LIN {X 0,Y 573.119,Z 536.24,A -85,B 0,C 180,E1 -2257.22,E2 -2257.22} C_VEL
LIN {X 0,Y 573.2,Z 527.994,A -85,B 0,C 180,E1 -2258.283,E2 -2258.283} C_VEL
LIN {X 0,Y 573.286,Z 519.543,A -85,B 0,C 180,E1 -2259.17,E2 -2259.17} C_VEL
LIN {X 0,Y 573.411,Z 509.104,A -85,B 0,C 180,E1 -2260.058,E2 -2260.058} C_VEL
LIN {X 0,Y 573.557,Z 497.409,A -85,B 0,C 180,E1 -2260.854,E2 -2260.854} C_VEL
LIN {X 0,Y 573.652,Z 486.296,A -85,B 0,C 180,E1 -2261.447,E2 -2261.447} C_VEL
LIN {X 0,Y 573.693,Z 474.485,A -85,B 0,C 180,E1 -2261.93,E2 -2261.93} C_VEL
LIN {X 0,Y 573.817,Z 461.452,A -85,B 0,C 180,E1 -2262.309,E2 -2262.309} C_VEL
LIN {X 0,Y 573.865,Z 449.117,A -85,B 0,C 180,E1 -2262.532,E2 -2262.532} C_VEL
LIN {X 0,Y 573.918,Z 350.087,A -85,B 0,C 180,E1 -2263.778,E2 -2263.778} C_VEL
LIN {X 0,Y 573.419,Z 346.442,A -85,B 0,C 180,E1 -2263.85,E2 -2263.85} C_VEL
LIN {X 0,Y 573.59,Z 325.392,A -85,B 0,C 180,E1 -2266.726,E2 -2266.726} C_VEL
LIN {X 0,Y 573.813,Z 304.327,A -85,B 0,C 180,E1 -2269.645,E2 -2269.645} C_VEL
LIN {X 0,Y 574.01,Z 285.256,A -85,B 0,C 180,E1 -2272.306,E2 -2272.306} C_VEL
LIN {X 0,Y 574.012,Z 277.944,A -85,B 0,C 180,E1 -2273.325,E2 -2273.325} C_VEL
LIN {X 0,Y 573.226,Z 274.085,A -85,B 0,C 180,E1 -2273.913,E2 -2273.913} C_VEL
LIN {X 0,Y 573.199,Z 274.087,A -85,B 0,C 180,E1 -2276.484,E2 -2276.484} C_VEL
LIN {X 0,Y 573.238,Z 274.076,A -85,B 0,C 180,E1 -2279.367,E2 -2279.367} C_VEL
LIN {X 0,Y 573.248,Z 274.082,A -85,B 0,C 180,E1 -2282.227,E2 -2282.227} C_VEL
LIN {X 0,Y 573.202,Z 274.08,A -85,B 0,C 180,E1 -2285.188,E2 -2285.188} C_VEL
LIN {X 0,Y 573.227,Z 274.077,A -85,B 0,C 180,E1 -2287.808,E2 -2287.808} C_VEL
LIN {X 0,Y 573.243,Z 274.082,A -85,B 0,C 180,E1 -2290.525,E2 -2290.525} C_VEL
LIN {X 0,Y 573.229,Z 274.075,A -85,B 0,C 180,E1 -2293.359,E2 -2293.359} C_VEL
LIN {X 0,Y 573.236,Z 274.082,A -85,B 0,C 180,E1 -2296.331,E2 -2296.331} C_VEL
LIN {X 0,Y 573.226,Z 274.085,A -85,B 0,C 180,E1 -2298.543,E2 -2298.543} C_VEL
LIN {X 0,Y 573.241,Z 274.074,A -85,B 0,C 180,E1 -2301.298,E2 -2301.298} C_VEL
LIN {X 0,Y 573.211,Z 274.079,A -85,B 0,C 180,E1 -2304.018,E2 -2304.018} C_VEL
LIN {X 0,Y 573.236,Z 274.083,A -85,B 0,C 180,E1 -2306.516,E2 -2306.516} C_VEL
LIN {X 0,Y 573.229,Z 274.077,A -85,B 0,C 180,E1 -2309.117,E2 -2309.117} C_VEL
LIN {X 0,Y 573.248,Z 274.073,A -85,B 0,C 180,E1 -2311.971,E2 -2311.971} C_VEL
LIN {X 0,Y 573.245,Z 274.082,A -85,B 0,C 180,E1 -2314.59,E2 -2314.59} C_VEL
LIN {X 0,Y 573.234,Z 274.074,A -85,B 0,C 180,E1 -2317.662,E2 -2317.662} C_VEL
LIN {X 0,Y 573.276,Z 274.079,A -85,B 0,C 180,E1 -2320.728,E2 -2320.728} C_VEL
LIN {X 0,Y 573.256,Z 274.071,A -85,B 0,C 180,E1 -2323.622,E2 -2323.622} C_VEL
LIN {X 0,Y 573.235,Z 274.08,A -85,B 0,C 180,E1 -2326.53,E2 -2326.53} C_VEL
LIN {X 0,Y 573.26,Z 274.08,A -85,B 0,C 180,E1 -2328.745,E2 -2328.745} C_VEL
LIN {X 0,Y 573.282,Z 274.068,A -85,B 0,C 180,E1 -2331.541,E2 -2331.541} C_VEL
LIN {X 0,Y 573.288,Z 274.07,A -85,B 0,C 180,E1 -2334.372,E2 -2334.372} C_VEL
LIN {X 0,Y 573.31,Z 274.065,A -85,B 0,C 180,E1 -2337.893,E2 -2337.893} C_VEL
LIN {X 0,Y 573.33,Z 274.068,A -85,B 0,C 180,E1 -2340.703,E2 -2340.703} C_VEL
LIN {X 0,Y 573.303,Z 274.074,A -85,B 0,C 180,E1 -2342.811,E2 -2342.811} C_VEL
LIN {X 0,Y 573.286,Z 274.069,A -85,B 0,C 180,E1 -2345.628,E2 -2345.628} C_VEL
LIN {X 0,Y 573.286,Z 274.07,A -85,B 0,C 180,E1 -2348.46,E2 -2348.46} C_VEL
LIN {X 0,Y 573.269,Z 274.076,A -85,B 0,C 180,E1 -2351.312,E2 -2351.312} C_VEL
LIN {X 0,Y 573.279,Z 274.069,A -85,B 0,C 180,E1 -2354.425,E2 -2354.425} C_VEL
LIN {X 0,Y 573.256,Z 274.081,A -85,B 0,C 180,E1 -2357.112,E2 -2357.112} C_VEL
LIN {X 0,Y 573.24,Z 274.073,A -85,B 0,C 180,E1 -2360.077,E2 -2360.077} C_VEL
LIN {X 0,Y 573.231,Z 274.075,A -85,B 0,C 180,E1 -2362.338,E2 -2362.338} C_VEL
LIN {X 0,Y 573.243,Z 274.074,A -85,B 0,C 180,E1 -2364.388,E2 -2364.388} C_VEL
LIN {X 0,Y 572.622,Z 274.158,A -85,B 0,C 180,E1 -2364.974,E2 -2364.974} C_VEL
LIN {X 0,Y 569.784,Z 274.516,A -85,B 0,C 180,E1 -2365.926,E2 -2365.926} C_VEL
LIN {X 0,Y 567.35,Z 274.82,A -85,B 0,C 180,E1 -2366.691,E2 -2366.691} C_VEL
LIN {X 0,Y 566.288,Z 274.949,A -85,B 0,C 180,E1 -2367.282,E2 -2367.282} C_VEL
LIN {X 0,Y 566.195,Z 274.957,A -85,B 0,C 180,E1 -2367.483,E2 -2367.483} C_VEL
LIN {X 0,Y 566.194,Z 274.954,A -85,B 0,C 180,E1 -2369.77,E2 -2369.77} C_VEL
LIN {X 0,Y 566.199,Z 274.95,A -85,B 0,C 180,E1 -2372.43,E2 -2372.43} C_VEL
LIN {X 0,Y 566.193,Z 274.957,A -85,B 0,C 180,E1 -2374.992,E2 -2374.992} C_VEL
LIN {X 0,Y 566.194,Z 274.958,A -85,B 0,C 180,E1 -2377.462,E2 -2377.462} C_VEL
LIN {X 0,Y 566.205,Z 274.95,A -85,B 0,C 180,E1 -2380.2,E2 -2380.2} C_VEL
LIN {X 0,Y 566.18,Z 274.958,A -85,B 0,C 180,E1 -2383.057,E2 -2383.057} C_VEL
LIN {X 0,Y 566.157,Z 274.958,A -85,B 0,C 180,E1 -2386.054,E2 -2386.054} C_VEL
LIN {X 0,Y 566.157,Z 274.958,A -85,B 0,C 180,E1 -2388.859,E2 -2388.859} C_VEL
LIN {X 0,Y 566.201,Z 274.961,A -85,B 0,C 180,E1 -2391.444,E2 -2391.444} C_VEL
LIN {X 0,Y 566.143,Z 274.958,A -85,B 0,C 180,E1 -2394.307,E2 -2394.307} C_VEL
LIN {X 0,Y 566.194,Z 274.954,A -85,B 0,C 180,E1 -2396.897,E2 -2396.897} C_VEL
LIN {X 0,Y 566.166,Z 274.964,A -85,B 0,C 180,E1 -2399.407,E2 -2399.407} C_VEL
LIN {X 0,Y 566.198,Z 274.956,A -85,B 0,C 180,E1 -2402.586,E2 -2402.586} C_VEL
LIN {X 0,Y 566.328,Z 280.666,A -85,B 0,C 180,E1 -2403.664,E2 -2403.664} C_VEL
LIN {X 0,Y 566.236,Z 295.178,A -85,B 0,C 180,E1 -2406.405,E2 -2406.405} C_VEL
LIN {X 0,Y 566.225,Z 298.604,A -85,B 0,C 180,E1 -2407.047,E2 -2407.047} C_VEL
LIN {X 0,Y 567.18,Z 304.563,A -85,B 0,C 180,E1 -2407.157,E2 -2407.157} C_VEL
LIN {X 0,Y 566.919,Z 405.543,A -85,B 0,C 180,E1 -2408.459,E2 -2408.459} C_VEL
LIN {X 0,Y 566.843,Z 419.197,A -85,B 0,C 180,E1 -2408.793,E2 -2408.793} C_VEL
LIN {X 0,Y 566.723,Z 431.898,A -85,B 0,C 180,E1 -2409.256,E2 -2409.256} C_VEL
LIN {X 0,Y 566.555,Z 444.148,A -85,B 0,C 180,E1 -2409.865,E2 -2409.865} C_VEL
LIN {X 0,Y 566.418,Z 455.088,A -85,B 0,C 180,E1 -2410.562,E2 -2410.562} C_VEL
LIN {X 0,Y 566.299,Z 465.233,A -85,B 0,C 180,E1 -2411.364,E2 -2411.364} C_VEL
LIN {X 0,Y 566.183,Z 474.756,A -85,B 0,C 180,E1 -2412.295,E2 -2412.295} C_VEL
LIN {X 0,Y 566.05,Z 483.938,A -85,B 0,C 180,E1 -2413.408,E2 -2413.408} C_VEL
LIN {X 0,Y 566.009,Z 491.238,A -85,B 0,C 180,E1 -2414.517,E2 -2414.517} C_VEL
LIN {X 0,Y 565.941,Z 496.998,A -85,B 0,C 180,E1 -2415.62,E2 -2415.62} C_VEL
LIN {X 0,Y 565.928,Z 501.492,A -85,B 0,C 180,E1 -2416.719,E2 -2416.719} C_VEL
LIN {X 0,Y 565.894,Z 504.853,A -85,B 0,C 180,E1 -2417.812,E2 -2417.812} C_VEL
LIN {X 0,Y 565.904,Z 507.1,A -85,B 0,C 180,E1 -2418.847,E2 -2418.847} C_VEL
LIN {X 0,Y 565.882,Z 508.554,A -85,B 0,C 180,E1 -2419.987,E2 -2419.987} C_VEL
LIN {X 0,Y 565.852,Z 508.921,A -85,B 0,C 180,E1 -2421.429,E2 -2421.429} C_VEL
LIN {X 0,Y 565.879,Z 508.522,A -85,B 0,C 180,E1 -2422.148,E2 -2422.148} C_VEL
LIN {X 0,Y 565.921,Z 506.681,A -85,B 0,C 180,E1 -2423.466,E2 -2423.466} C_VEL
LIN {X 0,Y 565.916,Z 503.806,A -85,B 0,C 180,E1 -2424.656,E2 -2424.656} C_VEL
LIN {X 0,Y 565.957,Z 500.162,A -85,B 0,C 180,E1 -2425.728,E2 -2425.728} C_VEL
LIN {X 0,Y 565.954,Z 495.423,A -85,B 0,C 180,E1 -2426.797,E2 -2426.797} C_VEL
LIN {X 0,Y 566.008,Z 488.339,A -85,B 0,C 180,E1 -2428.044,E2 -2428.044} C_VEL
LIN {X 0,Y 566.12,Z 480.648,A -85,B 0,C 180,E1 -2429.111,E2 -2429.111} C_VEL
LIN {X 0,Y 566.205,Z 471.063,A -85,B 0,C 180,E1 -2430.178,E2 -2430.178} C_VEL
LIN {X 0,Y 566.328,Z 461.195,A -85,B 0,C 180,E1 -2431.067,E2 -2431.067} C_VEL
LIN {X 0,Y 566.445,Z 450.086,A -85,B 0,C 180,E1 -2431.867,E2 -2431.867} C_VEL
LIN {X 0,Y 566.588,Z 439.243,A -85,B 0,C 180,E1 -2432.489,E2 -2432.489} C_VEL
LIN {X 0,Y 566.702,Z 427.292,A -85,B 0,C 180,E1 -2433.022,E2 -2433.022} C_VEL
LIN {X 0,Y 566.816,Z 414.954,A -85,B 0,C 180,E1 -2433.421,E2 -2433.421} C_VEL
LIN {X 0,Y 566.89,Z 402.186,A -85,B 0,C 180,E1 -2433.688,E2 -2433.688} C_VEL
LIN {X 0,Y 567.102,Z 303.98,A -85,B 0,C 180,E1 -2434.942,E2 -2434.942} C_VEL
LIN {X 0,Y 566.257,Z 298.554,A -85,B 0,C 180,E1 -2435.051,E2 -2435.051} C_VEL
LIN {X 0,Y 566.353,Z 283.716,A -85,B 0,C 180,E1 -2437.846,E2 -2437.846} C_VEL
LIN {X 0,Y 566.213,Z 275.181,A -85,B 0,C 180,E1 -2439.466,E2 -2439.466} C_VEL
LIN {X 0,Y 566.169,Z 274.959,A -85,B 0,C 180,E1 -2439.648,E2 -2439.648} C_VEL
LIN {X 0,Y 566.185,Z 274.958,A -85,B 0,C 180,E1 -2442.183,E2 -2442.183} C_VEL
LIN {X 0,Y 566.194,Z 274.954,A -85,B 0,C 180,E1 -2445.11,E2 -2445.11} C_VEL
LIN {X 0,Y 566.175,Z 274.955,A -85,B 0,C 180,E1 -2448.079,E2 -2448.079} C_VEL
LIN {X 0,Y 566.208,Z 274.953,A -85,B 0,C 180,E1 -2450.338,E2 -2450.338} C_VEL
LIN {X 0,Y 566.171,Z 274.957,A -85,B 0,C 180,E1 -2453.28,E2 -2453.28} C_VEL
LIN {X 0,Y 566.178,Z 274.953,A -85,B 0,C 180,E1 -2455.751,E2 -2455.751} C_VEL
LIN {X 0,Y 566.157,Z 274.956,A -85,B 0,C 180,E1 -2458.192,E2 -2458.192} C_VEL
LIN {X 0,Y 566.182,Z 274.962,A -85,B 0,C 180,E1 -2461.074,E2 -2461.074} C_VEL
LIN {X 0,Y 566.202,Z 274.951,A -85,B 0,C 180,E1 -2463.732,E2 -2463.732} C_VEL
LIN {X 0,Y 566.185,Z 274.954,A -85,B 0,C 180,E1 -2466.572,E2 -2466.572} C_VEL
LIN {X 0,Y 566.21,Z 274.952,A -85,B 0,C 180,E1 -2469.684,E2 -2469.684} C_VEL
LIN {X 0,Y 566.183,Z 274.959,A -85,B 0,C 180,E1 -2473.056,E2 -2473.056} C_VEL
LIN {X 0,Y 566.16,Z 274.956,A -85,B 0,C 180,E1 -2476.053,E2 -2476.053} C_VEL
LIN {X 0,Y 566.159,Z 274.958,A -85,B 0,C 180,E1 -2478.858,E2 -2478.858} C_VEL
LIN {X 0,Y 566.203,Z 274.961,A -85,B 0,C 180,E1 -2481.444,E2 -2481.444} C_VEL
LIN {X 0,Y 566.146,Z 274.957,A -85,B 0,C 180,E1 -2484.306,E2 -2484.306} C_VEL
LIN {X 0,Y 566.199,Z 274.951,A -85,B 0,C 180,E1 -2486.896,E2 -2486.896} C_VEL
LIN {X 0,Y 566.171,Z 274.961,A -85,B 0,C 180,E1 -2489.406,E2 -2489.406} C_VEL
LIN {X 0,Y 566.193,Z 274.959,A -85,B 0,C 180,E1 -2491.856,E2 -2491.856} C_VEL
LIN {X 0,Y 566.183,Z 274.953,A -85,B 0,C 180,E1 -2494.979,E2 -2494.979} C_VEL
LIN {X 0,Y 566.191,Z 274.956,A -85,B 0,C 180,E1 -2498.137,E2 -2498.137} C_VEL
LIN {X 0,Y 566.236,Z 274.946,A -85,B 0,C 180,E1 -2500.614,E2 -2500.614} C_VEL
LIN {X 0,Y 566.169,Z 274.957,A -85,B 0,C 180,E1 -2503.411,E2 -2503.411} C_VEL
LIN {X 0,Y 566.226,Z 274.952,A -85,B 0,C 180,E1 -2505.626,E2 -2505.626} C_VEL
LIN {X 0,Y 566.194,Z 274.952,A -85,B 0,C 180,E1 -2508.699,E2 -2508.699} C_VEL
LIN {X 0,Y 566.198,Z 274.952,A -85,B 0,C 180,E1 -2511.434,E2 -2511.434} C_VEL
LIN {X 0,Y 566.242,Z 274.953,A -85,B 0,C 180,E1 -2514.301,E2 -2514.301} C_VEL
LIN {X 0,Y 566.279,Z 274.945,A -85,B 0,C 180,E1 -2517.866,E2 -2517.866} C_VEL
LIN {X 0,Y 566.289,Z 274.943,A -85,B 0,C 180,E1 -2520.711,E2 -2520.711} C_VEL
LIN {X 0,Y 566.249,Z 274.947,A -85,B 0,C 180,E1 -2522.846,E2 -2522.846} C_VEL
LIN {X 0,Y 566.232,Z 274.947,A -85,B 0,C 180,E1 -2525.698,E2 -2525.698} C_VEL
LIN {X 0,Y 566.192,Z 274.96,A -85,B 0,C 180,E1 -2528.566,E2 -2528.566} C_VEL
LIN {X 0,Y 566.197,Z 274.951,A -85,B 0,C 180,E1 -2531.455,E2 -2531.455} C_VEL
LIN {X 0,Y 566.218,Z 274.957,A -85,B 0,C 180,E1 -2534.498,E2 -2534.498} C_VEL
LIN {X 0,Y 566.176,Z 274.954,A -85,B 0,C 180,E1 -2537.332,E2 -2537.332} C_VEL
LIN {X 0,Y 566.205,Z 274.954,A -85,B 0,C 180,E1 -2540.337,E2 -2540.337} C_VEL
LIN {X 0,Y 566.169,Z 274.957,A -85,B 0,C 180,E1 -2543.279,E2 -2543.279} C_VEL
LIN {X 0,Y 566.174,Z 274.953,A -85,B 0,C 180,E1 -2545.751,E2 -2545.751} C_VEL
LIN {X 0,Y 566.154,Z 274.957,A -85,B 0,C 180,E1 -2548.192,E2 -2548.192} C_VEL
LIN {X 0,Y 566.179,Z 274.962,A -85,B 0,C 180,E1 -2551.073,E2 -2551.073} C_VEL
LIN {X 0,Y 566.199,Z 274.951,A -85,B 0,C 180,E1 -2553.731,E2 -2553.731} C_VEL
LIN {X 0,Y 566.183,Z 274.955,A -85,B 0,C 180,E1 -2556.571,E2 -2556.571} C_VEL
LIN {X 0,Y 566.208,Z 274.952,A -85,B 0,C 180,E1 -2559.684,E2 -2559.684} C_VEL
LIN {X 0,Y 566.181,Z 274.96,A -85,B 0,C 180,E1 -2563.056,E2 -2563.056} C_VEL
LIN {X 0,Y 566.158,Z 274.956,A -85,B 0,C 180,E1 -2566.053,E2 -2566.053} C_VEL
LIN {X 0,Y 566.156,Z 274.958,A -85,B 0,C 180,E1 -2568.858,E2 -2568.858} C_VEL
LIN {X 0,Y 566.201,Z 274.961,A -85,B 0,C 180,E1 -2571.443,E2 -2571.443} C_VEL
LIN {X 0,Y 566.144,Z 274.957,A -85,B 0,C 180,E1 -2574.306,E2 -2574.306} C_VEL
LIN {X 0,Y 566.197,Z 274.952,A -85,B 0,C 180,E1 -2576.896,E2 -2576.896} C_VEL
LIN {X 0,Y 566.169,Z 274.961,A -85,B 0,C 180,E1 -2579.406,E2 -2579.406} C_VEL
LIN {X 0,Y 566.191,Z 274.959,A -85,B 0,C 180,E1 -2581.856,E2 -2581.856} C_VEL
LIN {X 0,Y 566.181,Z 274.956,A -85,B 0,C 180,E1 -2584.979,E2 -2584.979} C_VEL
LIN {X 0,Y 566.223,Z 275.057,A -85,B 0,C 180,E1 -2585.966,E2 -2585.966} C_VEL
LIN {X 0,Y 567.099,Z 280.881,A -85,B 0,C 180,E1 -2586.829,E2 -2586.829} C_VEL
LIN {X 0,Y 566.937,Z 299.897,A -85,B 0,C 180,E1 -2589.5,E2 -2589.5} C_VEL
LIN {X 0,Y 566.706,Z 318.68,A -85,B 0,C 180,E1 -2592.125,E2 -2592.125} C_VEL
LIN {X 0,Y 566.465,Z 341.208,A -85,B 0,C 180,E1 -2595.255,E2 -2595.255} C_VEL
LIN {X 0,Y 566.413,Z 346.518,A -85,B 0,C 180,E1 -2595.986,E2 -2595.986} C_VEL
LIN {X 0,Y 567.167,Z 353.204,A -85,B 0,C 180,E1 -2596.095,E2 -2596.095} C_VEL
LIN {X 0,Y 566.929,Z 454.923,A -85,B 0,C 180,E1 -2597.402,E2 -2597.402} C_VEL
LIN {X 0,Y 566.839,Z 468.203,A -85,B 0,C 180,E1 -2597.718,E2 -2597.718} C_VEL
LIN {X 0,Y 566.749,Z 480.365,A -85,B 0,C 180,E1 -2598.148,E2 -2598.148} C_VEL
LIN {X 0,Y 566.628,Z 492.144,A -85,B 0,C 180,E1 -2598.708,E2 -2598.708} C_VEL
LIN {X 0,Y 566.454,Z 504.192,A -85,B 0,C 180,E1 -2599.455,E2 -2599.455} C_VEL
LIN {X 0,Y 566.322,Z 514.597,A -85,B 0,C 180,E1 -2600.265,E2 -2600.265} C_VEL
LIN {X 0,Y 566.207,Z 523.108,A -85,B 0,C 180,E1 -2601.074,E2 -2601.074} C_VEL
LIN {X 0,Y 566.113,Z 530.957,A -85,B 0,C 180,E1 -2601.971,E2 -2601.971} C_VEL
LIN {X 0,Y 566.004,Z 538.619,A -85,B 0,C 180,E1 -2603.046,E2 -2603.046} C_VEL
LIN {X 0,Y 566.004,Z 545.677,A -85,B 0,C 180,E1 -2604.299,E2 -2604.299} C_VEL
LIN {X 0,Y 565.933,Z 550.371,A -85,B 0,C 180,E1 -2605.37,E2 -2605.37} C_VEL
LIN {X 0,Y 565.927,Z 553.956,A -85,B 0,C 180,E1 -2606.44,E2 -2606.44} C_VEL
LIN {X 0,Y 565.878,Z 555.807,A -85,B 0,C 180,E1 -2607.152,E2 -2607.152} C_VEL
LIN {X 0,Y 565.845,Z 558.184,A -85,B 0,C 180,E1 -2608.576,E2 -2608.576} C_VEL
LIN {X 0,Y 565.839,Z 559,A -85,B 0,C 180,E1 -2610,E2 -2610} C_VEL
LIN {X 0,Y 565.845,Z 558.186,A -85,B 0,C 180,E1 -2611.423,E2 -2611.423} C_VEL
LIN {X 0,Y 565.878,Z 555.811,A -85,B 0,C 180,E1 -2612.847,E2 -2612.847} C_VEL
LIN {X 0,Y 565.926,Z 552.897,A -85,B 0,C 180,E1 -2613.916,E2 -2613.916} C_VEL
LIN {X 0,Y 565.878,Z 548.95,A -85,B 0,C 180,E1 -2614.987,E2 -2614.987} C_VEL
LIN {X 0,Y 566.002,Z 543.869,A -85,B 0,C 180,E1 -2616.058,E2 -2616.058} C_VEL
LIN {X 0,Y 566.039,Z 537.471,A -85,B 0,C 180,E1 -2617.132,E2 -2617.132} C_VEL
LIN {X 0,Y 566.133,Z 529.482,A -85,B 0,C 180,E1 -2618.207,E2 -2618.207} C_VEL
LIN {X 0,Y 566.228,Z 521.339,A -85,B 0,C 180,E1 -2619.105,E2 -2619.105} C_VEL
LIN {X 0,Y 566.34,Z 511.405,A -85,B 0,C 180,E1 -2620.004,E2 -2620.004} C_VEL
LIN {X 0,Y 566.552,Z 500.309,A -85,B 0,C 180,E1 -2620.806,E2 -2620.806} C_VEL
LIN {X 0,Y 566.64,Z 489.184,A -85,B 0,C 180,E1 -2621.446,E2 -2621.446} C_VEL
LIN {X 0,Y 566.756,Z 476.993,A -85,B 0,C 180,E1 -2621.987,E2 -2621.987} C_VEL
LIN {X 0,Y 566.858,Z 464.194,A -85,B 0,C 180,E1 -2622.394,E2 -2622.394} C_VEL
LIN {X 0,Y 566.951,Z 450.632,A -85,B 0,C 180,E1 -2622.665,E2 -2622.665} C_VEL
LIN {X 0,Y 567.042,Z 350.756,A -85,B 0,C 180,E1 -2623.94,E2 -2623.94} C_VEL
LIN {X 0,Y 566.433,Z 346.442,A -85,B 0,C 180,E1 -2624.024,E2 -2624.024} C_VEL
LIN {X 0,Y 566.63,Z 324.131,A -85,B 0,C 180,E1 -2627.114,E2 -2627.114} C_VEL
LIN {X 0,Y 566.893,Z 303.963,A -85,B 0,C 180,E1 -2629.933,E2 -2629.933} C_VEL
LIN {X 0,Y 567.151,Z 282.169,A -85,B 0,C 180,E1 -2632.975,E2 -2632.975} C_VEL
LIN {X 0,Y 566.801,Z 278.191,A -85,B 0,C 180,E1 -2633.551,E2 -2633.551} C_VEL
LIN {X 0,Y 566.197,Z 274.961,A -85,B 0,C 180,E1 -2634.034,E2 -2634.034} C_VEL
LIN {X 0,Y 566.169,Z 274.961,A -85,B 0,C 180,E1 -2636.651,E2 -2636.651} C_VEL
LIN {X 0,Y 566.171,Z 274.958,A -85,B 0,C 180,E1 -2638.954,E2 -2638.954} C_VEL
LIN {X 0,Y 566.188,Z 274.954,A -85,B 0,C 180,E1 -2641.422,E2 -2641.422} C_VEL
LIN {X 0,Y 566.195,Z 274.957,A -85,B 0,C 180,E1 -2643.956,E2 -2643.956} C_VEL
LIN {X 0,Y 566.18,Z 274.961,A -85,B 0,C 180,E1 -2646.571,E2 -2646.571} C_VEL
LIN {X 0,Y 566.209,Z 274.95,A -85,B 0,C 180,E1 -2649.274,E2 -2649.274} C_VEL
LIN {X 0,Y 566.185,Z 274.957,A -85,B 0,C 180,E1 -2652.089,E2 -2652.089} C_VEL
LIN {X 0,Y 566.166,Z 274.957,A -85,B 0,C 180,E1 -2655.036,E2 -2655.036} C_VEL
LIN {X 0,Y 566.186,Z 274.954,A -85,B 0,C 180,E1 -2657.91,E2 -2657.91} C_VEL
LIN {X 0,Y 566.216,Z 274.955,A -85,B 0,C 180,E1 -2660.726,E2 -2660.726} C_VEL
LIN {X 0,Y 566.182,Z 274.953,A -85,B 0,C 180,E1 -2663.788,E2 -2663.788} C_VEL
LIN {X 0,Y 566.195,Z 274.956,A -85,B 0,C 180,E1 -2666.268,E2 -2666.268} C_VEL
LIN {X 0,Y 566.191,Z 274.956,A -85,B 0,C 180,E1 -2668.923,E2 -2668.923} C_VEL
LIN {X 0,Y 566.209,Z 274.949,A -85,B 0,C 180,E1 -2671.857,E2 -2671.857} C_VEL
LIN {X 0,Y 566.206,Z 274.953,A -85,B 0,C 180,E1 -2674.251,E2 -2674.251} C_VEL
LIN {X 0,Y 566.169,Z 274.965,A -85,B 0,C 180,E1 -2676.718,E2 -2676.718} C_VEL
LIN {X 0,Y 566.211,Z 274.948,A -85,B 0,C 180,E1 -2679.663,E2 -2679.663} C_VEL
LIN {X 0,Y 566.198,Z 274.96,A -85,B 0,C 180,E1 -2682.668,E2 -2682.668} C_VEL
LIN {X 0,Y 566.232,Z 274.947,A -85,B 0,C 180,E1 -2685.627,E2 -2685.627} C_VEL
LIN {X 0,Y 566.232,Z 274.954,A -85,B 0,C 180,E1 -2688.675,E2 -2688.675} C_VEL
LIN {X 0,Y 566.226,Z 274.948,A -85,B 0,C 180,E1 -2691.434,E2 -2691.434} C_VEL
LIN {X 0,Y 566.256,Z 274.946,A -85,B 0,C 180,E1 -2694.302,E2 -2694.302} C_VEL
LIN {X 0,Y 566.281,Z 274.94,A -85,B 0,C 180,E1 -2697.866,E2 -2697.866} C_VEL
LIN {X 0,Y 566.301,Z 274.944,A -85,B 0,C 180,E1 -2700.711,E2 -2700.711} C_VEL
LIN {X 0,Y 566.269,Z 274.95,A -85,B 0,C 180,E1 -2702.846,E2 -2702.846} C_VEL
LIN {X 0,Y 566.254,Z 274.944,A -85,B 0,C 180,E1 -2705.699,E2 -2705.699} C_VEL
LIN {X 0,Y 566.229,Z 274.95,A -85,B 0,C 180,E1 -2708.566,E2 -2708.566} C_VEL
LIN {X 0,Y 566.24,Z 274.949,A -85,B 0,C 180,E1 -2711.455,E2 -2711.455} C_VEL
LIN {X 0,Y 566.232,Z 274.948,A -85,B 0,C 180,E1 -2714.507,E2 -2714.507} C_VEL
LIN {X 0,Y 566.196,Z 274.957,A -85,B 0,C 180,E1 -2717.332,E2 -2717.332} C_VEL
LIN {X 0,Y 566.206,Z 274.95,A -85,B 0,C 180,E1 -2720.338,E2 -2720.338} C_VEL
LIN {X 0,Y 566.165,Z 274.963,A -85,B 0,C 180,E1 -2723.281,E2 -2723.281} C_VEL
LIN {X 0,Y 566.205,Z 274.952,A -85,B 0,C 180,E1 -2725.75,E2 -2725.75} C_VEL
LIN {X 0,Y 566.195,Z 274.957,A -85,B 0,C 180,E1 -2727.483,E2 -2727.483} C_VEL
LIN {X 0,Y 565.508,Z 275.039,A -85,B 0,C 180,E1 -2728.076,E2 -2728.076} C_VEL
LIN {X 0,Y 562.643,Z 275.401,A -85,B 0,C 180,E1 -2729.04,E2 -2729.04} C_VEL
LIN {X 0,Y 560.237,Z 275.696,A -85,B 0,C 180,E1 -2729.816,E2 -2729.816} C_VEL
LIN {X 0,Y 559.212,Z 275.822,A -85,B 0,C 180,E1 -2730.414,E2 -2730.414} C_VEL
LIN {X 0,Y 559.132,Z 275.832,A -85,B 0,C 180,E1 -2730.617,E2 -2730.617} C_VEL
LIN {X 0,Y 559.15,Z 275.83,A -85,B 0,C 180,E1 -2732.716,E2 -2732.716} C_VEL
LIN {X 0,Y 559.134,Z 275.84,A -85,B 0,C 180,E1 -2735.324,E2 -2735.324} C_VEL
LIN {X 0,Y 559.128,Z 275.832,A -85,B 0,C 180,E1 -2738.019,E2 -2738.019} C_VEL
LIN {X 0,Y 559.152,Z 275.831,A -85,B 0,C 180,E1 -2740.813,E2 -2740.813} C_VEL
LIN {X 0,Y 559.108,Z 275.839,A -85,B 0,C 180,E1 -2743.738,E2 -2743.738} C_VEL
LIN {X 0,Y 559.109,Z 275.835,A -85,B 0,C 180,E1 -2746.264,E2 -2746.264} C_VEL
LIN {X 0,Y 559.142,Z 275.833,A -85,B 0,C 180,E1 -2748.952,E2 -2748.952} C_VEL
LIN {X 0,Y 559.168,Z 275.833,A -85,B 0,C 180,E1 -2751.193,E2 -2751.193} C_VEL
LIN {X 0,Y 559.117,Z 275.838,A -85,B 0,C 180,E1 -2753.788,E2 -2753.788} C_VEL
LIN {X 0,Y 559.146,Z 275.83,A -85,B 0,C 180,E1 -2756.425,E2 -2756.425} C_VEL
LIN {X 0,Y 559.147,Z 275.833,A -85,B 0,C 180,E1 -2758.981,E2 -2758.981} C_VEL
LIN {X 0,Y 559.15,Z 275.835,A -85,B 0,C 180,E1 -2762.287,E2 -2762.287} C_VEL
LIN {X 0,Y 559.185,Z 275.921,A -85,B 0,C 180,E1 -2762.619,E2 -2762.619} C_VEL
LIN {X 0,Y 559.288,Z 283.029,A -85,B 0,C 180,E1 -2763.909,E2 -2763.909} C_VEL
LIN {X 0,Y 559.187,Z 298.612,A -85,B 0,C 180,E1 -2766.869,E2 -2766.869} C_VEL
LIN {X 0,Y 560.327,Z 306.565,A -85,B 0,C 180,E1 -2767.01,E2 -2767.01} C_VEL
LIN {X 0,Y 560.001,Z 405.224,A -85,B 0,C 180,E1 -2768.295,E2 -2768.295} C_VEL
LIN {X 0,Y 559.929,Z 418.809,A -85,B 0,C 180,E1 -2768.628,E2 -2768.628} C_VEL
LIN {X 0,Y 559.761,Z 431.314,A -85,B 0,C 180,E1 -2769.082,E2 -2769.082} C_VEL
LIN {X 0,Y 559.594,Z 443.721,A -85,B 0,C 180,E1 -2769.7,E2 -2769.7} C_VEL
LIN {X 0,Y 559.431,Z 455.052,A -85,B 0,C 180,E1 -2770.427,E2 -2770.427} C_VEL
LIN {X 0,Y 559.283,Z 466.003,A -85,B 0,C 180,E1 -2771.311,E2 -2771.311} C_VEL
LIN {X 0,Y 559.136,Z 475.378,A -85,B 0,C 180,E1 -2772.254,E2 -2772.254} C_VEL
LIN {X 0,Y 559.015,Z 483.057,A -85,B 0,C 180,E1 -2773.193,E2 -2773.193} C_VEL
LIN {X 0,Y 558.904,Z 490.544,A -85,B 0,C 180,E1 -2774.315,E2 -2774.315} C_VEL
LIN {X 0,Y 558.851,Z 496.975,A -85,B 0,C 180,E1 -2775.545,E2 -2775.545} C_VEL
LIN {X 0,Y 558.807,Z 502.36,A -85,B 0,C 180,E1 -2776.916,E2 -2776.916} C_VEL
LIN {X 0,Y 558.805,Z 504.566,A -85,B 0,C 180,E1 -2777.655,E2 -2777.655} C_VEL
LIN {X 0,Y 558.802,Z 507.093,A -85,B 0,C 180,E1 -2778.816,E2 -2778.816} C_VEL
LIN {X 0,Y 558.779,Z 508.463,A -85,B 0,C 180,E1 -2779.859,E2 -2779.859} C_VEL
LIN {X 0,Y 558.74,Z 508.906,A -85,B 0,C 180,E1 -2780.589,E2 -2780.589} C_VEL
LIN {X 0,Y 558.797,Z 508.598,A -85,B 0,C 180,E1 -2782.048,E2 -2782.048} C_VEL
LIN {X 0,Y 558.797,Z 507.857,A -85,B 0,C 180,E1 -2782.775,E2 -2782.775} C_VEL
LIN {X 0,Y 558.828,Z 506.673,A -85,B 0,C 180,E1 -2783.501,E2 -2783.501} C_VEL
LIN {X 0,Y 558.839,Z 504.14,A -85,B 0,C 180,E1 -2784.588,E2 -2784.588} C_VEL
LIN {X 0,Y 558.861,Z 500.61,A -85,B 0,C 180,E1 -2785.673,E2 -2785.673} C_VEL
LIN {X 0,Y 558.874,Z 495.991,A -85,B 0,C 180,E1 -2786.756,E2 -2786.756} C_VEL
LIN {X 0,Y 558.918,Z 489.042,A -85,B 0,C 180,E1 -2788.019,E2 -2788.019} C_VEL
LIN {X 0,Y 559.063,Z 481.538,A -85,B 0,C 180,E1 -2789.1,E2 -2789.1} C_VEL
LIN {X 0,Y 559.122,Z 473.911,A -85,B 0,C 180,E1 -2790,E2 -2790} C_VEL
LIN {X 0,Y 559.298,Z 463.584,A -85,B 0,C 180,E1 -2790.99,E2 -2790.99} C_VEL
LIN {X 0,Y 559.414,Z 453.119,A -85,B 0,C 180,E1 -2791.8,E2 -2791.8} C_VEL
LIN {X 0,Y 559.586,Z 441.428,A -85,B 0,C 180,E1 -2792.52,E2 -2792.52} C_VEL
LIN {X 0,Y 559.722,Z 428.982,A -85,B 0,C 180,E1 -2793.104,E2 -2793.104} C_VEL
LIN {X 0,Y 559.877,Z 415.817,A -85,B 0,C 180,E1 -2793.554,E2 -2793.554} C_VEL
LIN {X 0,Y 559.986,Z 403.68,A -85,B 0,C 180,E1 -2793.823,E2 -2793.823} C_VEL
LIN {X 0,Y 560.219,Z 304.777,A -85,B 0,C 180,E1 -2795.106,E2 -2795.106} C_VEL
LIN {X 0,Y 559.229,Z 298.57,A -85,B 0,C 180,E1 -2795.228,E2 -2795.228} C_VEL
LIN {X 0,Y 559.35,Z 282.346,A -85,B 0,C 180,E1 -2798.308,E2 -2798.308} C_VEL
LIN {X 0,Y 559.143,Z 275.835,A -85,B 0,C 180,E1 -2799.542,E2 -2799.542} C_VEL
LIN {X 0,Y 559.155,Z 275.836,A -85,B 0,C 180,E1 -2802.338,E2 -2802.338} C_VEL
LIN {X 0,Y 559.143,Z 275.831,A -85,B 0,C 180,E1 -2805.305,E2 -2805.305} C_VEL
LIN {X 0,Y 559.128,Z 275.831,A -85,B 0,C 180,E1 -2807.558,E2 -2807.558} C_VEL
LIN {X 0,Y 559.179,Z 275.832,A -85,B 0,C 180,E1 -2810.605,E2 -2810.605} C_VEL
LIN {X 0,Y 559.124,Z 275.832,A -85,B 0,C 180,E1 -2813.718,E2 -2813.718} C_VEL
LIN {X 0,Y 559.148,Z 275.829,A -85,B 0,C 180,E1 -2816.099,E2 -2816.099} C_VEL
LIN {X 0,Y 559.116,Z 275.836,A -85,B 0,C 180,E1 -2818.533,E2 -2818.533} C_VEL
LIN {X 0,Y 559.13,Z 275.837,A -85,B 0,C 180,E1 -2821.269,E2 -2821.269} C_VEL
LIN {X 0,Y 559.159,Z 275.827,A -85,B 0,C 180,E1 -2823.947,E2 -2823.947} C_VEL
LIN {X 0,Y 559.136,Z 275.841,A -85,B 0,C 180,E1 -2827.109,E2 -2827.109} C_VEL
LIN {X 0,Y 559.155,Z 275.829,A -85,B 0,C 180,E1 -2829.94,E2 -2829.94} C_VEL
LIN {X 0,Y 559.129,Z 275.841,A -85,B 0,C 180,E1 -2833.194,E2 -2833.194} C_VEL
LIN {X 0,Y 559.128,Z 275.835,A -85,B 0,C 180,E1 -2835.764,E2 -2835.764} C_VEL
LIN {X 0,Y 559.106,Z 275.834,A -85,B 0,C 180,E1 -2838.224,E2 -2838.224} C_VEL
LIN {X 0,Y 559.171,Z 275.83,A -85,B 0,C 180,E1 -2841.065,E2 -2841.065} C_VEL
LIN {X 0,Y 559.121,Z 275.838,A -85,B 0,C 180,E1 -2843.787,E2 -2843.787} C_VEL
LIN {X 0,Y 559.15,Z 275.829,A -85,B 0,C 180,E1 -2846.424,E2 -2846.424} C_VEL
LIN {X 0,Y 559.152,Z 275.83,A -85,B 0,C 180,E1 -2848.98,E2 -2848.98} C_VEL
LIN {X 0,Y 559.138,Z 275.84,A -85,B 0,C 180,E1 -2851.626,E2 -2851.626} C_VEL
LIN {X 0,Y 559.142,Z 275.829,A -85,B 0,C 180,E1 -2854.822,E2 -2854.822} C_VEL
LIN {X 0,Y 559.139,Z 275.84,A -85,B 0,C 180,E1 -2857.847,E2 -2857.847} C_VEL
LIN {X 0,Y 559.197,Z 275.824,A -85,B 0,C 180,E1 -2860.494,E2 -2860.494} C_VEL
LIN {X 0,Y 559.146,Z 275.83,A -85,B 0,C 180,E1 -2863.196,E2 -2863.196} C_VEL
LIN {X 0,Y 559.158,Z 275.834,A -85,B 0,C 180,E1 -2866.183,E2 -2866.183} C_VEL
LIN {X 0,Y 559.168,Z 275.826,A -85,B 0,C 180,E1 -2869.133,E2 -2869.133} C_VEL
LIN {X 0,Y 559.146,Z 275.839,A -85,B 0,C 180,E1 -2872.053,E2 -2872.053} C_VEL
LIN {X 0,Y 559.23,Z 275.819,A -85,B 0,C 180,E1 -2874.953,E2 -2874.953} C_VEL
LIN {X 0,Y 559.25,Z 275.82,A -85,B 0,C 180,E1 -2877.839,E2 -2877.839} C_VEL
LIN {X 0,Y 559.26,Z 275.818,A -85,B 0,C 180,E1 -2880.72,E2 -2880.72} C_VEL
LIN {X 0,Y 559.215,Z 275.823,A -85,B 0,C 180,E1 -2882.881,E2 -2882.881} C_VEL
LIN {X 0,Y 559.203,Z 275.823,A -85,B 0,C 180,E1 -2885.77,E2 -2885.77} C_VEL
LIN {X 0,Y 559.157,Z 275.835,A -85,B 0,C 180,E1 -2888.675,E2 -2888.675} C_VEL
LIN {X 0,Y 559.16,Z 275.827,A -85,B 0,C 180,E1 -2891.601,E2 -2891.601} C_VEL
LIN {X 0,Y 559.165,Z 275.837,A -85,B 0,C 180,E1 -2894.579,E2 -2894.579} C_VEL
LIN {X 0,Y 559.125,Z 275.832,A -85,B 0,C 180,E1 -2897.558,E2 -2897.558} C_VEL
LIN {X 0,Y 559.176,Z 275.833,A -85,B 0,C 180,E1 -2900.605,E2 -2900.605} C_VEL
LIN {X 0,Y 559.121,Z 275.832,A -85,B 0,C 180,E1 -2903.718,E2 -2903.718} C_VEL
LIN {X 0,Y 559.144,Z 275.83,A -85,B 0,C 180,E1 -2906.099,E2 -2906.099} C_VEL
LIN {X 0,Y 559.113,Z 275.837,A -85,B 0,C 180,E1 -2908.532,E2 -2908.532} C_VEL
LIN {X 0,Y 559.127,Z 275.837,A -85,B 0,C 180,E1 -2911.269,E2 -2911.269} C_VEL
LIN {X 0,Y 559.156,Z 275.828,A -85,B 0,C 180,E1 -2913.947,E2 -2913.947} C_VEL
LIN {X 0,Y 559.133,Z 275.841,A -85,B 0,C 180,E1 -2917.109,E2 -2917.109} C_VEL
LIN {X 0,Y 559.152,Z 275.829,A -85,B 0,C 180,E1 -2919.94,E2 -2919.94} C_VEL
LIN {X 0,Y 559.127,Z 275.842,A -85,B 0,C 180,E1 -2923.194,E2 -2923.194} C_VEL
LIN {X 0,Y 559.125,Z 275.835,A -85,B 0,C 180,E1 -2925.764,E2 -2925.764} C_VEL
LIN {X 0,Y 559.103,Z 275.834,A -85,B 0,C 180,E1 -2928.224,E2 -2928.224} C_VEL
LIN {X 0,Y 559.169,Z 275.831,A -85,B 0,C 180,E1 -2931.065,E2 -2931.065} C_VEL
LIN {X 0,Y 559.119,Z 275.837,A -85,B 0,C 180,E1 -2933.787,E2 -2933.787} C_VEL
LIN {X 0,Y 559.148,Z 275.829,A -85,B 0,C 180,E1 -2936.424,E2 -2936.424} C_VEL
LIN {X 0,Y 559.15,Z 275.83,A -85,B 0,C 180,E1 -2938.98,E2 -2938.98} C_VEL
LIN {X 0,Y 559.136,Z 275.841,A -85,B 0,C 180,E1 -2941.625,E2 -2941.625} C_VEL
LIN {X 0,Y 559.14,Z 275.833,A -85,B 0,C 180,E1 -2944.822,E2 -2944.822} C_VEL
LIN {X 0,Y 559.181,Z 275.926,A -85,B 0,C 180,E1 -2945.817,E2 -2945.817} C_VEL
LIN {X 0,Y 560.165,Z 282.008,A -85,B 0,C 180,E1 -2946.732,E2 -2946.732} C_VEL
LIN {X 0,Y 559.969,Z 300.946,A -85,B 0,C 180,E1 -2949.425,E2 -2949.425} C_VEL
LIN {X 0,Y 559.723,Z 319.906,A -85,B 0,C 180,E1 -2952.083,E2 -2952.083} C_VEL
LIN {X 0,Y 559.445,Z 342.955,A -85,B 0,C 180,E1 -2955.31,E2 -2955.31} C_VEL
LIN {X 0,Y 559.412,Z 346.435,A -85,B 0,C 180,E1 -2955.796,E2 -2955.796} C_VEL
LIN {X 0,Y 560.293,Z 353.204,A -85,B 0,C 180,E1 -2955.92,E2 -2955.92} C_VEL
LIN {X 0,Y 560.016,Z 454.923,A -85,B 0,C 180,E1 -2957.244,E2 -2957.244} C_VEL
LIN {X 0,Y 559.906,Z 468.202,A -85,B 0,C 180,E1 -2957.564,E2 -2957.564} C_VEL
LIN {X 0,Y 559.797,Z 480.367,A -85,B 0,C 180,E1 -2957.999,E2 -2957.999} C_VEL
LIN {X 0,Y 559.669,Z 491.802,A -85,B 0,C 180,E1 -2958.547,E2 -2958.547} C_VEL
LIN {X 0,Y 559.496,Z 502.898,A -85,B 0,C 180,E1 -2959.231,E2 -2959.231} C_VEL
LIN {X 0,Y 559.311,Z 513.533,A -85,B 0,C 180,E1 -2960.05,E2 -2960.05} C_VEL
LIN {X 0,Y 559.162,Z 523.109,A -85,B 0,C 180,E1 -2960.96,E2 -2960.96} C_VEL
LIN {X 0,Y 559.05,Z 530.957,A -85,B 0,C 180,E1 -2961.869,E2 -2961.869} C_VEL
LIN {X 0,Y 558.944,Z 538.62,A -85,B 0,C 180,E1 -2962.958,E2 -2962.958} C_VEL
LIN {X 0,Y 558.935,Z 545.677,A -85,B 0,C 180,E1 -2964.226,E2 -2964.226} C_VEL
LIN {X 0,Y 558.826,Z 550.371,A -85,B 0,C 180,E1 -2965.311,E2 -2965.311} C_VEL
LIN {X 0,Y 558.836,Z 553.957,A -85,B 0,C 180,E1 -2966.394,E2 -2966.394} C_VEL
LIN {X 0,Y 558.799,Z 555.806,A -85,B 0,C 180,E1 -2967.116,E2 -2967.116} C_VEL
LIN {X 0,Y 558.745,Z 558.183,A -85,B 0,C 180,E1 -2968.558,E2 -2968.558} C_VEL
LIN {X 0,Y 558.74,Z 559,A -85,B 0,C 180,E1 -2970,E2 -2970} C_VEL
LIN {X 0,Y 558.745,Z 558.185,A -85,B 0,C 180,E1 -2971.441,E2 -2971.441} C_VEL
LIN {X 0,Y 558.799,Z 555.811,A -85,B 0,C 180,E1 -2972.883,E2 -2972.883} C_VEL
LIN {X 0,Y 558.844,Z 552.897,A -85,B 0,C 180,E1 -2973.966,E2 -2973.966} C_VEL
LIN {X 0,Y 558.798,Z 548.95,A -85,B 0,C 180,E1 -2975.05,E2 -2975.05} C_VEL
LIN {X 0,Y 558.919,Z 543.869,A -85,B 0,C 180,E1 -2976.135,E2 -2976.135} C_VEL
LIN {X 0,Y 558.976,Z 537.47,A -85,B 0,C 180,E1 -2977.222,E2 -2977.222} C_VEL
LIN {X 0,Y 559.098,Z 529.481,A -85,B 0,C 180,E1 -2978.311,E2 -2978.311} C_VEL
LIN {X 0,Y 559.184,Z 521.339,A -85,B 0,C 180,E1 -2979.221,E2 -2979.221} C_VEL
LIN {X 0,Y 559.341,Z 511.404,A -85,B 0,C 180,E1 -2980.131,E2 -2980.131} C_VEL
LIN {X 0,Y 559.561,Z 500.386,A -85,B 0,C 180,E1 -2980.937,E2 -2980.937} C_VEL
LIN {X 0,Y 559.67,Z 488.468,A -85,B 0,C 180,E1 -2981.627,E2 -2981.627} C_VEL
LIN {X 0,Y 559.801,Z 475.781,A -85,B 0,C 180,E1 -2982.185,E2 -2982.185} C_VEL
LIN {X 0,Y 559.952,Z 462.364,A -85,B 0,C 180,E1 -2982.596,E2 -2982.596} C_VEL
LIN {X 0,Y 560.022,Z 449.117,A -85,B 0,C 180,E1 -2982.847,E2 -2982.847} C_VEL
LIN {X 0,Y 560.235,Z 352.22,A -85,B 0,C 180,E1 -2984.094,E2 -2984.094} C_VEL
LIN {X 0,Y 559.438,Z 346.442,A -85,B 0,C 180,E1 -2984.203,E2 -2984.203} C_VEL
LIN {X 0,Y 559.647,Z 324.796,A -85,B 0,C 180,E1 -2987.237,E2 -2987.237} C_VEL
LIN {X 0,Y 559.922,Z 304.964,A -85,B 0,C 180,E1 -2990,E2 -2990} C_VEL
LIN {X 0,Y 560.218,Z 283.218,A -85,B 0,C 180,E1 -2993.075,E2 -2993.075} C_VEL
LIN {X 0,Y 559.493,Z 277.672,A -85,B 0,C 180,E1 -2993.897,E2 -2993.897} C_VEL
LIN {X 0,Y 559.156,Z 275.839,A -85,B 0,C 180,E1 -2994.208,E2 -2994.208} C_VEL
LIN {X 0,Y 559.113,Z 275.837,A -85,B 0,C 180,E1 -2996.905,E2 -2996.905} C_VEL
LIN {X 0,Y 559.115,Z 275.836,A -85,B 0,C 180,E1 -2999.355,E2 -2999.355} C_VEL
LIN {X 0,Y 559.162,Z 275.833,A -85,B 0,C 180,E1 -3001.862,E2 -3001.862} C_VEL
LIN {X 0,Y 559.135,Z 275.841,A -85,B 0,C 180,E1 -3004.445,E2 -3004.445} C_VEL
LIN {X 0,Y 559.129,Z 275.833,A -85,B 0,C 180,E1 -3007.109,E2 -3007.109} C_VEL
LIN {X 0,Y 559.156,Z 275.831,A -85,B 0,C 180,E1 -3009.941,E2 -3009.941} C_VEL
LIN {X 0,Y 559.153,Z 275.834,A -85,B 0,C 180,E1 -3012.744,E2 -3012.744} C_VEL
LIN {X 0,Y 559.146,Z 275.83,A -85,B 0,C 180,E1 -3015.761,E2 -3015.761} C_VEL
LIN {X 0,Y 559.16,Z 275.834,A -85,B 0,C 180,E1 -3018.229,E2 -3018.229} C_VEL
LIN {X 0,Y 559.173,Z 275.827,A -85,B 0,C 180,E1 -3021.191,E2 -3021.191} C_VEL
LIN {X 0,Y 559.137,Z 275.831,A -85,B 0,C 180,E1 -3023.789,E2 -3023.789} C_VEL
LIN {X 0,Y 559.146,Z 275.836,A -85,B 0,C 180,E1 -3026.424,E2 -3026.424} C_VEL
LIN {X 0,Y 559.155,Z 275.832,A -85,B 0,C 180,E1 -3028.981,E2 -3028.981} C_VEL
LIN {X 0,Y 559.165,Z 275.826,A -85,B 0,C 180,E1 -3031.619,E2 -3031.619} C_VEL
LIN {X 0,Y 559.175,Z 275.826,A -85,B 0,C 180,E1 -3033.903,E2 -3033.903} C_VEL
LIN {X 0,Y 559.138,Z 275.837,A -85,B 0,C 180,E1 -3036.571,E2 -3036.571} C_VEL
LIN {X 0,Y 559.177,Z 275.825,A -85,B 0,C 180,E1 -3039.395,E2 -3039.395} C_VEL
LIN {X 0,Y 559.144,Z 275.83,A -85,B 0,C 180,E1 -3041.686,E2 -3041.686} C_VEL
LIN {X 0,Y 559.167,Z 275.826,A -85,B 0,C 180,E1 -3043.948,E2 -3043.948} C_VEL
LIN {X 0,Y 559.172,Z 275.828,A -85,B 0,C 180,E1 -3046.184,E2 -3046.184} C_VEL
LIN {X 0,Y 559.191,Z 275.829,A -85,B 0,C 180,E1 -3049.134,E2 -3049.134} C_VEL
LIN {X 0,Y 559.201,Z 275.822,A -85,B 0,C 180,E1 -3052.054,E2 -3052.054} C_VEL
LIN {X 0,Y 559.249,Z 275.825,A -85,B 0,C 180,E1 -3054.953,E2 -3054.953} C_VEL
LIN {X 0,Y 559.252,Z 275.816,A -85,B 0,C 180,E1 -3057.84,E2 -3057.84} C_VEL
LIN {X 0,Y 559.271,Z 275.82,A -85,B 0,C 180,E1 -3060.72,E2 -3060.72} C_VEL
LIN {X 0,Y 559.236,Z 275.827,A -85,B 0,C 180,E1 -3062.882,E2 -3062.882} C_VEL
LIN {X 0,Y 559.224,Z 275.82,A -85,B 0,C 180,E1 -3065.77,E2 -3065.77} C_VEL
LIN {X 0,Y 559.188,Z 275.828,A -85,B 0,C 180,E1 -3068.675,E2 -3068.675} C_VEL
LIN {X 0,Y 559.203,Z 275.824,A -85,B 0,C 180,E1 -3071.601,E2 -3071.601} C_VEL
LIN {X 0,Y 559.198,Z 275.825,A -85,B 0,C 180,E1 -3074.596,E2 -3074.596} C_VEL
LIN {X 0,Y 559.139,Z 275.833,A -85,B 0,C 180,E1 -3077.558,E2 -3077.558} C_VEL
LIN {X 0,Y 559.164,Z 275.828,A -85,B 0,C 180,E1 -3079.838,E2 -3079.838} C_VEL
LIN {X 0,Y 559.138,Z 275.83,A -85,B 0,C 180,E1 -3082.153,E2 -3082.153} C_VEL
LIN {X 0,Y 559.173,Z 275.834,A -85,B 0,C 180,E1 -3085.299,E2 -3085.299} C_VEL
LIN {X 0,Y 559.146,Z 275.832,A -85,B 0,C 180,E1 -3087.714,E2 -3087.714} C_VEL
LIN {X 0,Y 559.132,Z 275.832,A -85,B 0,C 180,E1 -3090.617,E2 -3090.617} C_VEL
LIN {X 0,Y 558.471,Z 275.924,A -85,B 0,C 180,E1 -3091.219,E2 -3091.219} C_VEL
LIN {X 0,Y 555.609,Z 276.277,A -85,B 0,C 180,E1 -3092.195,E2 -3092.195} C_VEL
LIN {X 0,Y 553.193,Z 276.576,A -85,B 0,C 180,E1 -3092.98,E2 -3092.98} C_VEL
LIN {X 0,Y 552.167,Z 276.704,A -85,B 0,C 180,E1 -3093.587,E2 -3093.587} C_VEL
LIN {X 0,Y 552.09,Z 276.709,A -85,B 0,C 180,E1 -3093.792,E2 -3093.792} C_VEL
LIN {X 0,Y 552.104,Z 276.708,A -85,B 0,C 180,E1 -3096.748,E2 -3096.748} C_VEL
LIN {X 0,Y 552.125,Z 276.711,A -85,B 0,C 180,E1 -3099.528,E2 -3099.528} C_VEL
LIN {X 0,Y 552.106,Z 276.707,A -85,B 0,C 180,E1 -3102.428,E2 -3102.428} C_VEL
LIN {X 0,Y 552.075,Z 276.718,A -85,B 0,C 180,E1 -3105.561,E2 -3105.561} C_VEL
LIN {X 0,Y 552.076,Z 276.711,A -85,B 0,C 180,E1 -3108.551,E2 -3108.551} C_VEL
LIN {X 0,Y 552.111,Z 276.715,A -85,B 0,C 180,E1 -3111.411,E2 -3111.411} C_VEL
LIN {X 0,Y 552.071,Z 276.711,A -85,B 0,C 180,E1 -3114.156,E2 -3114.156} C_VEL
LIN {X 0,Y 552.105,Z 276.708,A -85,B 0,C 180,E1 -3116.814,E2 -3116.814} C_VEL
LIN {X 0,Y 552.091,Z 276.718,A -85,B 0,C 180,E1 -3119.391,E2 -3119.391} C_VEL
LIN {X 0,Y 552.13,Z 276.829,A -85,B 0,C 180,E1 -3122.599,E2 -3122.599} C_VEL
LIN {X 0,Y 552.251,Z 284.31,A -85,B 0,C 180,E1 -3123.957,E2 -3123.957} C_VEL
LIN {X 0,Y 552.15,Z 298.292,A -85,B 0,C 180,E1 -3126.6,E2 -3126.6} C_VEL
LIN {X 0,Y 552.161,Z 298.818,A -85,B 0,C 180,E1 -3126.694,E2 -3126.694} C_VEL
LIN {X 0,Y 553.452,Z 306.612,A -85,B 0,C 180,E1 -3126.831,E2 -3126.831} C_VEL
LIN {X 0,Y 553.076,Z 405.308,A -85,B 0,C 180,E1 -3128.134,E2 -3128.134} C_VEL
LIN {X 0,Y 552.995,Z 418.872,A -85,B 0,C 180,E1 -3128.472,E2 -3128.472} C_VEL
LIN {X 0,Y 552.807,Z 431.851,A -85,B 0,C 180,E1 -3128.952,E2 -3128.952} C_VEL
LIN {X 0,Y 552.625,Z 443.29,A -85,B 0,C 180,E1 -3129.53,E2 -3129.53} C_VEL
LIN {X 0,Y 552.439,Z 455.055,A -85,B 0,C 180,E1 -3130.291,E2 -3130.291} C_VEL
LIN {X 0,Y 552.254,Z 465.733,A -85,B 0,C 180,E1 -3131.161,E2 -3131.161} C_VEL
LIN {X 0,Y 552.082,Z 475.998,A -85,B 0,C 180,E1 -3132.211,E2 -3132.211} C_VEL
LIN {X 0,Y 551.935,Z 484.939,A -85,B 0,C 180,E1 -3133.352,E2 -3133.352} C_VEL
LIN {X 0,Y 551.843,Z 492.005,A -85,B 0,C 180,E1 -3134.488,E2 -3134.488} C_VEL
LIN {X 0,Y 551.775,Z 498.109,A -85,B 0,C 180,E1 -3135.732,E2 -3135.732} C_VEL
LIN {X 0,Y 551.727,Z 501.961,A -85,B 0,C 180,E1 -3136.745,E2 -3136.745} C_VEL
LIN {X 0,Y 551.707,Z 504.251,A -85,B 0,C 180,E1 -3137.494,E2 -3137.494} C_VEL
LIN {X 0,Y 551.713,Z 507.076,A -85,B 0,C 180,E1 -3138.776,E2 -3138.776} C_VEL
LIN {X 0,Y 551.676,Z 508.339,A -85,B 0,C 180,E1 -3139.727,E2 -3139.727} C_VEL
LIN {X 0,Y 551.659,Z 508.876,A -85,B 0,C 180,E1 -3140.467,E2 -3140.467} C_VEL
LIN {X 0,Y 551.671,Z 508.971,A -85,B 0,C 180,E1 -3141.207,E2 -3141.207} C_VEL
LIN {X 0,Y 551.696,Z 508.674,A -85,B 0,C 180,E1 -3141.945,E2 -3141.945} C_VEL
LIN {X 0,Y 551.693,Z 507.989,A -85,B 0,C 180,E1 -3142.682,E2 -3142.682} C_VEL
LIN {X 0,Y 551.733,Z 506.733,A -85,B 0,C 180,E1 -3143.502,E2 -3143.502} C_VEL
LIN {X 0,Y 551.71,Z 503.412,A -85,B 0,C 180,E1 -3144.885,E2 -3144.885} C_VEL
LIN {X 0,Y 551.777,Z 499.637,A -85,B 0,C 180,E1 -3145.983,E2 -3145.983} C_VEL
LIN {X 0,Y 551.779,Z 494.759,A -85,B 0,C 180,E1 -3147.08,E2 -3147.08} C_VEL
LIN {X 0,Y 551.864,Z 488.631,A -85,B 0,C 180,E1 -3148.176,E2 -3148.176} C_VEL
LIN {X 0,Y 552.009,Z 481.03,A -85,B 0,C 180,E1 -3149.271,E2 -3149.271} C_VEL
LIN {X 0,Y 552.136,Z 471.524,A -85,B 0,C 180,E1 -3150.365,E2 -3150.365} C_VEL
LIN {X 0,Y 552.304,Z 461.749,A -85,B 0,C 180,E1 -3151.276,E2 -3151.276} C_VEL
LIN {X 0,Y 552.465,Z 450.814,A -85,B 0,C 180,E1 -3152.096,E2 -3152.096} C_VEL
LIN {X 0,Y 552.647,Z 438.412,A -85,B 0,C 180,E1 -3152.825,E2 -3152.825} C_VEL
LIN {X 0,Y 552.813,Z 426.192,A -85,B 0,C 180,E1 -3153.371,E2 -3153.371} C_VEL
LIN {X 0,Y 552.958,Z 413.219,A -85,B 0,C 180,E1 -3153.781,E2 -3153.781} C_VEL
LIN {X 0,Y 553.094,Z 400.763,A -85,B 0,C 180,E1 -3154.031,E2 -3154.031} C_VEL
LIN {X 0,Y 553.367,Z 305.775,A -85,B 0,C 180,E1 -3155.272,E2 -3155.272} C_VEL
LIN {X 0,Y 552.176,Z 298.698,A -85,B 0,C 180,E1 -3155.41,E2 -3155.41} C_VEL
LIN {X 0,Y 552.323,Z 282.822,A -85,B 0,C 180,E1 -3158.415,E2 -3158.415} C_VEL
LIN {X 0,Y 552.09,Z 276.714,A -85,B 0,C 180,E1 -3159.595,E2 -3159.595} C_VEL
LIN {X 0,Y 552.108,Z 276.708,A -85,B 0,C 180,E1 -3161.752,E2 -3161.752} C_VEL
LIN {X 0,Y 552.129,Z 276.712,A -85,B 0,C 180,E1 -3164.749,E2 -3164.749} C_VEL
LIN {X 0,Y 552.088,Z 276.708,A -85,B 0,C 180,E1 -3167.79,E2 -3167.79} C_VEL
LIN {X 0,Y 552.125,Z 276.705,A -85,B 0,C 180,E1 -3170.102,E2 -3170.102} C_VEL
LIN {X 0,Y 552.089,Z 276.712,A -85,B 0,C 180,E1 -3172.452,E2 -3172.452} C_VEL
LIN {X 0,Y 552.084,Z 276.712,A -85,B 0,C 180,E1 -3175.333,E2 -3175.333} C_VEL
LIN {X 0,Y 552.062,Z 276.712,A -85,B 0,C 180,E1 -3178.101,E2 -3178.101} C_VEL
LIN {X 0,Y 552.08,Z 276.713,A -85,B 0,C 180,E1 -3180.611,E2 -3180.611} C_VEL
LIN {X 0,Y 552.109,Z 276.714,A -85,B 0,C 180,E1 -3183.187,E2 -3183.187} C_VEL
LIN {X 0,Y 552.077,Z 276.71,A -85,B 0,C 180,E1 -3185.845,E2 -3185.845} C_VEL
LIN {X 0,Y 552.117,Z 276.706,A -85,B 0,C 180,E1 -3188.59,E2 -3188.59} C_VEL
LIN {X 0,Y 552.063,Z 276.718,A -85,B 0,C 180,E1 -3191.452,E2 -3191.452} C_VEL
LIN {X 0,Y 552.08,Z 276.71,A -85,B 0,C 180,E1 -3194.529,E2 -3194.529} C_VEL
LIN {X 0,Y 552.088,Z 276.715,A -85,B 0,C 180,E1 -3197.59,E2 -3197.59} C_VEL
LIN {X 0,Y 552.113,Z 276.705,A -85,B 0,C 180,E1 -3200.471,E2 -3200.471} C_VEL
LIN {X 0,Y 552.101,Z 276.714,A -85,B 0,C 180,E1 -3203.319,E2 -3203.319} C_VEL
LIN {X 0,Y 552.104,Z 276.71,A -85,B 0,C 180,E1 -3205.937,E2 -3205.937} C_VEL
LIN {X 0,Y 552.126,Z 276.703,A -85,B 0,C 180,E1 -3208.541,E2 -3208.541} C_VEL
LIN {X 0,Y 552.099,Z 276.713,A -85,B 0,C 180,E1 -3211.444,E2 -3211.444} C_VEL
LIN {X 0,Y 552.075,Z 276.711,A -85,B 0,C 180,E1 -3214.353,E2 -3214.353} C_VEL
LIN {X 0,Y 552.096,Z 276.707,A -85,B 0,C 180,E1 -3216.757,E2 -3216.757} C_VEL
LIN {X 0,Y 552.121,Z 276.705,A -85,B 0,C 180,E1 -3219.119,E2 -3219.119} C_VEL
LIN {X 0,Y 552.084,Z 276.712,A -85,B 0,C 180,E1 -3221.443,E2 -3221.443} C_VEL
LIN {X 0,Y 552.087,Z 276.715,A -85,B 0,C 180,E1 -3223.736,E2 -3223.736} C_VEL
LIN {X 0,Y 552.128,Z 276.714,A -85,B 0,C 180,E1 -3226.004,E2 -3226.004} C_VEL
LIN {X 0,Y 552.13,Z 276.703,A -85,B 0,C 180,E1 -3228.992,E2 -3228.992} C_VEL
LIN {X 0,Y 552.115,Z 276.712,A -85,B 0,C 180,E1 -3231.951,E2 -3231.951} C_VEL
LIN {X 0,Y 552.208,Z 276.694,A -85,B 0,C 180,E1 -3234.889,E2 -3234.889} C_VEL
LIN {X 0,Y 552.221,Z 276.695,A -85,B 0,C 180,E1 -3237.812,E2 -3237.812} C_VEL
LIN {X 0,Y 552.232,Z 276.694,A -85,B 0,C 180,E1 -3240.729,E2 -3240.729} C_VEL
LIN {X 0,Y 552.182,Z 276.698,A -85,B 0,C 180,E1 -3242.918,E2 -3242.918} C_VEL
LIN {X 0,Y 552.175,Z 276.699,A -85,B 0,C 180,E1 -3245.844,E2 -3245.844} C_VEL
LIN {X 0,Y 552.129,Z 276.708,A -85,B 0,C 180,E1 -3248.786,E2 -3248.786} C_VEL
LIN {X 0,Y 552.106,Z 276.706,A -85,B 0,C 180,E1 -3251.752,E2 -3251.752} C_VEL
LIN {X 0,Y 552.127,Z 276.711,A -85,B 0,C 180,E1 -3254.749,E2 -3254.749} C_VEL
LIN {X 0,Y 552.085,Z 276.709,A -85,B 0,C 180,E1 -3257.789,E2 -3257.789} C_VEL
LIN {X 0,Y 552.123,Z 276.705,A -85,B 0,C 180,E1 -3260.101,E2 -3260.101} C_VEL
LIN {X 0,Y 552.087,Z 276.713,A -85,B 0,C 180,E1 -3262.451,E2 -3262.451} C_VEL
LIN {X 0,Y 552.081,Z 276.712,A -85,B 0,C 180,E1 -3265.333,E2 -3265.333} C_VEL
LIN {X 0,Y 552.059,Z 276.712,A -85,B 0,C 180,E1 -3268.101,E2 -3268.101} C_VEL
LIN {X 0,Y 552.077,Z 276.714,A -85,B 0,C 180,E1 -3270.611,E2 -3270.611} C_VEL
LIN {X 0,Y 552.107,Z 276.713,A -85,B 0,C 180,E1 -3273.186,E2 -3273.186} C_VEL
LIN {X 0,Y 552.074,Z 276.71,A -85,B 0,C 180,E1 -3275.845,E2 -3275.845} C_VEL
LIN {X 0,Y 552.115,Z 276.707,A -85,B 0,C 180,E1 -3278.589,E2 -3278.589} C_VEL
LIN {X 0,Y 552.061,Z 276.718,A -85,B 0,C 180,E1 -3281.452,E2 -3281.452} C_VEL
LIN {X 0,Y 552.078,Z 276.71,A -85,B 0,C 180,E1 -3284.529,E2 -3284.529} C_VEL
LIN {X 0,Y 552.085,Z 276.714,A -85,B 0,C 180,E1 -3287.59,E2 -3287.59} C_VEL
LIN {X 0,Y 552.11,Z 276.705,A -85,B 0,C 180,E1 -3290.471,E2 -3290.471} C_VEL
LIN {X 0,Y 552.099,Z 276.715,A -85,B 0,C 180,E1 -3293.318,E2 -3293.318} C_VEL
LIN {X 0,Y 552.102,Z 276.71,A -85,B 0,C 180,E1 -3295.937,E2 -3295.937} C_VEL
LIN {X 0,Y 552.124,Z 276.704,A -85,B 0,C 180,E1 -3298.54,E2 -3298.54} C_VEL
LIN {X 0,Y 552.098,Z 276.715,A -85,B 0,C 180,E1 -3301.444,E2 -3301.444} C_VEL
LIN {X 0,Y 552.073,Z 276.715,A -85,B 0,C 180,E1 -3304.352,E2 -3304.352} C_VEL
LIN {X 0,Y 552.104,Z 276.789,A -85,B 0,C 180,E1 -3305.662,E2 -3305.662} C_VEL
LIN {X 0,Y 553.139,Z 282.429,A -85,B 0,C 180,E1 -3306.529,E2 -3306.529} C_VEL
LIN {X 0,Y 553.068,Z 296.559,A -85,B 0,C 180,E1 -3308.571,E2 -3308.571} C_VEL
LIN {X 0,Y 552.771,Z 315.541,A -85,B 0,C 180,E1 -3311.274,E2 -3311.274} C_VEL
LIN {X 0,Y 552.495,Z 334.463,A -85,B 0,C 180,E1 -3313.938,E2 -3313.938} C_VEL
LIN {X 0,Y 552.403,Z 346.516,A -85,B 0,C 180,E1 -3315.623,E2 -3315.623} C_VEL
LIN {X 0,Y 553.382,Z 354.271,A -85,B 0,C 180,E1 -3315.755,E2 -3315.755} C_VEL
LIN {X 0,Y 553.116,Z 454.923,A -85,B 0,C 180,E1 -3317.082,E2 -3317.082} C_VEL
LIN {X 0,Y 552.964,Z 468.201,A -85,B 0,C 180,E1 -3317.405,E2 -3317.405} C_VEL
LIN {X 0,Y 552.835,Z 480.357,A -85,B 0,C 180,E1 -3317.845,E2 -3317.845} C_VEL
LIN {X 0,Y 552.691,Z 492.651,A -85,B 0,C 180,E1 -3318.449,E2 -3318.449} C_VEL
LIN {X 0,Y 552.496,Z 504.187,A -85,B 0,C 180,E1 -3319.185,E2 -3319.185} C_VEL
LIN {X 0,Y 552.298,Z 514.6,A -85,B 0,C 180,E1 -3320.015,E2 -3320.015} C_VEL
LIN {X 0,Y 552.126,Z 523.109,A -85,B 0,C 180,E1 -3320.844,E2 -3320.844} C_VEL
LIN {X 0,Y 552.013,Z 530.957,A -85,B 0,C 180,E1 -3321.765,E2 -3321.765} C_VEL
LIN {X 0,Y 551.89,Z 538.619,A -85,B 0,C 180,E1 -3322.867,E2 -3322.867} C_VEL
LIN {X 0,Y 551.867,Z 545.677,A -85,B 0,C 180,E1 -3324.152,E2 -3324.152} C_VEL
LIN {X 0,Y 551.725,Z 550.371,A -85,B 0,C 180,E1 -3325.25,E2 -3325.25} C_VEL
LIN {X 0,Y 551.75,Z 553.957,A -85,B 0,C 180,E1 -3326.348,E2 -3326.348} C_VEL
LIN {X 0,Y 551.723,Z 555.806,A -85,B 0,C 180,E1 -3327.079,E2 -3327.079} C_VEL
LIN {X 0,Y 551.645,Z 558.182,A -85,B 0,C 180,E1 -3328.539,E2 -3328.539} C_VEL
LIN {X 0,Y 551.64,Z 559,A -85,B 0,C 180,E1 -3330,E2 -3330} C_VEL
LIN {X 0,Y 551.645,Z 558.185,A -85,B 0,C 180,E1 -3331.46,E2 -3331.46} C_VEL
LIN {X 0,Y 551.723,Z 555.811,A -85,B 0,C 180,E1 -3332.92,E2 -3332.92} C_VEL
LIN {X 0,Y 551.764,Z 552.897,A -85,B 0,C 180,E1 -3334.017,E2 -3334.017} C_VEL
LIN {X 0,Y 551.723,Z 548.95,A -85,B 0,C 180,E1 -3335.115,E2 -3335.115} C_VEL
LIN {X 0,Y 551.814,Z 543.129,A -85,B 0,C 180,E1 -3336.352,E2 -3336.352} C_VEL
LIN {X 0,Y 551.926,Z 536.239,A -85,B 0,C 180,E1 -3337.499,E2 -3337.499} C_VEL
LIN {X 0,Y 552.082,Z 527.995,A -85,B 0,C 180,E1 -3338.602,E2 -3338.602} C_VEL
LIN {X 0,Y 552.222,Z 519.544,A -85,B 0,C 180,E1 -3339.523,E2 -3339.523} C_VEL
LIN {X 0,Y 552.384,Z 509.098,A -85,B 0,C 180,E1 -3340.445,E2 -3340.445} C_VEL
LIN {X 0,Y 552.625,Z 498.197,A -85,B 0,C 180,E1 -3341.219,E2 -3341.219} C_VEL
LIN {X 0,Y 552.749,Z 487.414,A -85,B 0,C 180,E1 -3341.83,E2 -3341.83} C_VEL
LIN {X 0,Y 552.863,Z 475.777,A -85,B 0,C 180,E1 -3342.34,E2 -3342.34} C_VEL
LIN {X 0,Y 553.038,Z 462.363,A -85,B 0,C 180,E1 -3342.756,E2 -3342.756} C_VEL
LIN {X 0,Y 553.127,Z 449.117,A -85,B 0,C 180,E1 -3343.01,E2 -3343.01} C_VEL
LIN {X 0,Y 553.379,Z 353.301,A -85,B 0,C 180,E1 -3344.258,E2 -3344.258} C_VEL
LIN {X 0,Y 552.43,Z 346.442,A -85,B 0,C 180,E1 -3344.386,E2 -3344.386} C_VEL
LIN {X 0,Y 552.627,Z 326.013,A -85,B 0,C 180,E1 -3347.242,E2 -3347.242} C_VEL
LIN {X 0,Y 552.947,Z 304.611,A -85,B 0,C 180,E1 -3350.264,E2 -3350.264} C_VEL
LIN {X 0,Y 553.255,Z 284.18,A -85,B 0,C 180,E1 -3353.19,E2 -3353.19} C_VEL
LIN {X 0,Y 552.103,Z 276.717,A -85,B 0,C 180,E1 -3354.337,E2 -3354.337} C_VEL
LIN {X 0,Y 552.072,Z 276.713,A -85,B 0,C 180,E1 -3357.276,E2 -3357.276} C_VEL
LIN {X 0,Y 552.095,Z 276.717,A -85,B 0,C 180,E1 -3360.046,E2 -3360.046} C_VEL
LIN {X 0,Y 552.108,Z 276.711,A -85,B 0,C 180,E1 -3362.845,E2 -3362.845} C_VEL
LIN {X 0,Y 552.069,Z 276.713,A -85,B 0,C 180,E1 -3365.438,E2 -3365.438} C_VEL
LIN {X 0,Y 552.091,Z 276.711,A -85,B 0,C 180,E1 -3367.885,E2 -3367.885} C_VEL
LIN {X 0,Y 552.105,Z 276.716,A -85,B 0,C 180,E1 -3370.481,E2 -3370.481} C_VEL
LIN {X 0,Y 552.105,Z 276.707,A -85,B 0,C 180,E1 -3373.423,E2 -3373.423} C_VEL
LIN {X 0,Y 552.104,Z 276.716,A -85,B 0,C 180,E1 -3376.576,E2 -3376.576} C_VEL
LIN {X 0,Y 552.107,Z 276.706,A -85,B 0,C 180,E1 -3379.519,E2 -3379.519} C_VEL
LIN {X 0,Y 552.089,Z 276.715,A -85,B 0,C 180,E1 -3382.336,E2 -3382.336} C_VEL
LIN {X 0,Y 552.082,Z 276.711,A -85,B 0,C 180,E1 -3385.051,E2 -3385.051} C_VEL
LIN {X 0,Y 552.113,Z 276.705,A -85,B 0,C 180,E1 -3387.681,E2 -3387.681} C_VEL
LIN {X 0,Y 552.106,Z 276.71,A -85,B 0,C 180,E1 -3390.235,E2 -3390.235} C_VEL
LIN {X 0,Y 552.136,Z 276.707,A -85,B 0,C 180,E1 -3393,E2 -3393} C_VEL
LIN {X 0,Y 552.109,Z 276.707,A -85,B 0,C 180,E1 -3395.161,E2 -3395.161} C_VEL
LIN {X 0,Y 552.122,Z 276.708,A -85,B 0,C 180,E1 -3398.337,E2 -3398.337} C_VEL
LIN {X 0,Y 552.153,Z 276.708,A -85,B 0,C 180,E1 -3400.674,E2 -3400.674} C_VEL
LIN {X 0,Y 552.117,Z 276.704,A -85,B 0,C 180,E1 -3403.737,E2 -3403.737} C_VEL
LIN {X 0,Y 552.135,Z 276.703,A -85,B 0,C 180,E1 -3406.005,E2 -3406.005} C_VEL
LIN {X 0,Y 552.159,Z 276.707,A -85,B 0,C 180,E1 -3408.993,E2 -3408.993} C_VEL
LIN {X 0,Y 552.155,Z 276.699,A -85,B 0,C 180,E1 -3411.952,E2 -3411.952} C_VEL
LIN {X 0,Y 552.224,Z 276.701,A -85,B 0,C 180,E1 -3414.889,E2 -3414.889} C_VEL
LIN {X 0,Y 552.223,Z 276.692,A -85,B 0,C 180,E1 -3417.812,E2 -3417.812} C_VEL
LIN {X 0,Y 552.241,Z 276.696,A -85,B 0,C 180,E1 -3420.729,E2 -3420.729} C_VEL
LIN {X 0,Y 552.202,Z 276.704,A -85,B 0,C 180,E1 -3422.918,E2 -3422.918} C_VEL
LIN {X 0,Y 552.195,Z 276.695,A -85,B 0,C 180,E1 -3425.844,E2 -3425.844} C_VEL
LIN {X 0,Y 552.158,Z 276.706,A -85,B 0,C 180,E1 -3428.786,E2 -3428.786} C_VEL
LIN {X 0,Y 552.16,Z 276.7,A -85,B 0,C 180,E1 -3431.751,E2 -3431.751} C_VEL
LIN {X 0,Y 552.135,Z 276.707,A -85,B 0,C 180,E1 -3434.749,E2 -3434.749} C_VEL
LIN {X 0,Y 552.096,Z 276.708,A -85,B 0,C 180,E1 -3437.789,E2 -3437.789} C_VEL
LIN {X 0,Y 552.125,Z 276.704,A -85,B 0,C 180,E1 -3440.102,E2 -3440.102} C_VEL
LIN {X 0,Y 552.089,Z 276.709,A -85,B 0,C 180,E1 -3442.451,E2 -3442.451} C_VEL
LIN {X 0,Y 552.135,Z 276.71,A -85,B 0,C 180,E1 -3445.347,E2 -3445.347} C_VEL
LIN {X 0,Y 552.091,Z 276.708,A -85,B 0,C 180,E1 -3448.1,E2 -3448.1} C_VEL
LIN {X 0,Y 552.096,Z 276.709,A -85,B 0,C 180,E1 -3450.614,E2 -3450.614} C_VEL
LIN {X 0,Y 552.105,Z 276.714,A -85,B 0,C 180,E1 -3453.187,E2 -3453.187} C_VEL
LIN {X 0,Y 552.09,Z 276.709,A -85,B 0,C 180,E1 -3453.792,E2 -3453.792} C_VEL
LIN {X 0,Y 551.451,Z 276.79,A -85,B 0,C 180,E1 -3454.401,E2 -3454.401} C_VEL
LIN {X 0,Y 548.636,Z 277.147,A -85,B 0,C 180,E1 -3455.389,E2 -3455.389} C_VEL
LIN {X 0,Y 546.225,Z 277.443,A -85,B 0,C 180,E1 -3456.185,E2 -3456.185} C_VEL
LIN {X 0,Y 545.161,Z 277.574,A -85,B 0,C 180,E1 -3456.799,E2 -3456.799} C_VEL
LIN {X 0,Y 545.059,Z 277.589,A -85,B 0,C 180,E1 -3457.007,E2 -3457.007} C_VEL
LIN {X 0,Y 545.062,Z 277.584,A -85,B 0,C 180,E1 -3460.144,E2 -3460.144} C_VEL
LIN {X 0,Y 545.036,Z 277.589,A -85,B 0,C 180,E1 -3462.694,E2 -3462.694} C_VEL
LIN {X 0,Y 545.021,Z 277.596,A -85,B 0,C 180,E1 -3465.172,E2 -3465.172} C_VEL
LIN {X 0,Y 545.052,Z 277.589,A -85,B 0,C 180,E1 -3467.895,E2 -3467.895} C_VEL
LIN {X 0,Y 545.075,Z 277.585,A -85,B 0,C 180,E1 -3470.818,E2 -3470.818} C_VEL
LIN {X 0,Y 545.032,Z 277.595,A -85,B 0,C 180,E1 -3473.619,E2 -3473.619} C_VEL
LIN {X 0,Y 545.048,Z 277.587,A -85,B 0,C 180,E1 -3476.327,E2 -3476.327} C_VEL
LIN {X 0,Y 545.054,Z 277.589,A -85,B 0,C 180,E1 -3478.952,E2 -3478.952} C_VEL
LIN {X 0,Y 545.046,Z 277.598,A -85,B 0,C 180,E1 -3481.505,E2 -3481.505} C_VEL
LIN {X 0,Y 545.105,Z 277.693,A -85,B 0,C 180,E1 -3482.541,E2 -3482.541} C_VEL
LIN {X 0,Y 545.245,Z 284.544,A -85,B 0,C 180,E1 -3483.803,E2 -3483.803} C_VEL
LIN {X 0,Y 545.149,Z 297.679,A -85,B 0,C 180,E1 -3486.253,E2 -3486.253} C_VEL
LIN {X 0,Y 545.149,Z 298.903,A -85,B 0,C 180,E1 -3486.495,E2 -3486.495} C_VEL
LIN {X 0,Y 546.565,Z 307.808,A -85,B 0,C 180,E1 -3486.66,E2 -3486.66} C_VEL
LIN {X 0,Y 546.18,Z 405.548,A -85,B 0,C 180,E1 -3487.966,E2 -3487.966} C_VEL
LIN {X 0,Y 546.078,Z 419.149,A -85,B 0,C 180,E1 -3488.309,E2 -3488.309} C_VEL
LIN {X 0,Y 545.849,Z 431.534,A -85,B 0,C 180,E1 -3488.77,E2 -3488.77} C_VEL
LIN {X 0,Y 545.684,Z 443.096,A -85,B 0,C 180,E1 -3489.356,E2 -3489.356} C_VEL
LIN {X 0,Y 545.47,Z 453.882,A -85,B 0,C 180,E1 -3490.054,E2 -3490.054} C_VEL
LIN {X 0,Y 545.283,Z 464.495,A -85,B 0,C 180,E1 -3490.911,E2 -3490.911} C_VEL
LIN {X 0,Y 545.087,Z 473.281,A -85,B 0,C 180,E1 -3491.781,E2 -3491.781} C_VEL
LIN {X 0,Y 544.952,Z 481.301,A -85,B 0,C 180,E1 -3492.746,E2 -3492.746} C_VEL
LIN {X 0,Y 544.791,Z 489.093,A -85,B 0,C 180,E1 -3493.898,E2 -3493.898} C_VEL
LIN {X 0,Y 544.74,Z 495.32,A -85,B 0,C 180,E1 -3495.047,E2 -3495.047} C_VEL
LIN {X 0,Y 544.68,Z 500.204,A -85,B 0,C 180,E1 -3496.19,E2 -3496.19} C_VEL
LIN {X 0,Y 544.624,Z 503.91,A -85,B 0,C 180,E1 -3497.328,E2 -3497.328} C_VEL
LIN {X 0,Y 544.624,Z 507.058,A -85,B 0,C 180,E1 -3498.736,E2 -3498.736} C_VEL
LIN {X 0,Y 544.58,Z 508.211,A -85,B 0,C 180,E1 -3499.591,E2 -3499.591} C_VEL
LIN {X 0,Y 544.581,Z 508.81,A -85,B 0,C 180,E1 -3500.342,E2 -3500.342} C_VEL
LIN {X 0,Y 544.564,Z 508.996,A -85,B 0,C 180,E1 -3501.091,E2 -3501.091} C_VEL
LIN {X 0,Y 544.612,Z 508.749,A -85,B 0,C 180,E1 -3501.84,E2 -3501.84} C_VEL
LIN {X 0,Y 544.652,Z 507.09,A -85,B 0,C 180,E1 -3503.332,E2 -3503.332} C_VEL
LIN {X 0,Y 544.644,Z 505.642,A -85,B 0,C 180,E1 -3504.075,E2 -3504.075} C_VEL
LIN {X 0,Y 544.602,Z 502.668,A -85,B 0,C 180,E1 -3505.189,E2 -3505.189} C_VEL
LIN {X 0,Y 544.693,Z 498.651,A -85,B 0,C 180,E1 -3506.302,E2 -3506.302} C_VEL
LIN {X 0,Y 544.774,Z 492.49,A -85,B 0,C 180,E1 -3507.597,E2 -3507.597} C_VEL
LIN {X 0,Y 544.874,Z 485.807,A -85,B 0,C 180,E1 -3508.707,E2 -3508.707} C_VEL
LIN {X 0,Y 544.993,Z 477.584,A -85,B 0,C 180,E1 -3509.816,E2 -3509.816} C_VEL
LIN {X 0,Y 545.161,Z 469.158,A -85,B 0,C 180,E1 -3510.739,E2 -3510.739} C_VEL
LIN {X 0,Y 545.346,Z 458.805,A -85,B 0,C 180,E1 -3511.662,E2 -3511.662} C_VEL
LIN {X 0,Y 545.56,Z 447.16,A -85,B 0,C 180,E1 -3512.492,E2 -3512.492} C_VEL
LIN {X 0,Y 545.807,Z 435.428,A -85,B 0,C 180,E1 -3513.138,E2 -3513.138} C_VEL
LIN {X 0,Y 545.929,Z 423.303,A -85,B 0,C 180,E1 -3513.645,E2 -3513.645} C_VEL
LIN {X 0,Y 546.075,Z 410.844,A -85,B 0,C 180,E1 -3514.013,E2 -3514.013} C_VEL
LIN {X 0,Y 546.176,Z 396.197,A -85,B 0,C 180,E1 -3514.267,E2 -3514.267} C_VEL
LIN {X 0,Y 546.437,Z 306.085,A -85,B 0,C 180,E1 -3515.456,E2 -3515.456} C_VEL
LIN {X 0,Y 545.173,Z 298.892,A -85,B 0,C 180,E1 -3515.595,E2 -3515.595} C_VEL
LIN {X 0,Y 545.308,Z 283.45,A -85,B 0,C 180,E1 -3518.524,E2 -3518.524} C_VEL
LIN {X 0,Y 545.042,Z 277.593,A -85,B 0,C 180,E1 -3519.65,E2 -3519.65} C_VEL
LIN {X 0,Y 545.073,Z 277.586,A -85,B 0,C 180,E1 -3521.906,E2 -3521.906} C_VEL
LIN {X 0,Y 545.084,Z 277.586,A -85,B 0,C 180,E1 -3524.944,E2 -3524.944} C_VEL
LIN {X 0,Y 545.054,Z 277.585,A -85,B 0,C 180,E1 -3528.027,E2 -3528.027} C_VEL
LIN {X 0,Y 545.094,Z 277.583,A -85,B 0,C 180,E1 -3530.373,E2 -3530.373} C_VEL
LIN {X 0,Y 545.077,Z 277.582,A -85,B 0,C 180,E1 -3533.56,E2 -3533.56} C_VEL
LIN {X 0,Y 545.048,Z 277.594,A -85,B 0,C 180,E1 -3536.828,E2 -3536.828} C_VEL
LIN {X 0,Y 545.027,Z 277.592,A -85,B 0,C 180,E1 -3539.341,E2 -3539.341} C_VEL
LIN {X 0,Y 545.049,Z 277.585,A -85,B 0,C 180,E1 -3541.916,E2 -3541.916} C_VEL
LIN {X 0,Y 545.053,Z 277.587,A -85,B 0,C 180,E1 -3544.566,E2 -3544.566} C_VEL
LIN {X 0,Y 545.035,Z 277.594,A -85,B 0,C 180,E1 -3547.305,E2 -3547.305} C_VEL
LIN {X 0,Y 545.056,Z 277.584,A -85,B 0,C 180,E1 -3550.144,E2 -3550.144} C_VEL
LIN {X 0,Y 545.022,Z 277.596,A -85,B 0,C 180,E1 -3553.113,E2 -3553.113} C_VEL
LIN {X 0,Y 545.032,Z 277.587,A -85,B 0,C 180,E1 -3556.229,E2 -3556.229} C_VEL
LIN {X 0,Y 545.02,Z 277.591,A -85,B 0,C 180,E1 -3558.879,E2 -3558.879} C_VEL
LIN {X 0,Y 545.047,Z 277.59,A -85,B 0,C 180,E1 -3561.762,E2 -3561.762} C_VEL
LIN {X 0,Y 545.03,Z 277.587,A -85,B 0,C 180,E1 -3564.531,E2 -3564.531} C_VEL
LIN {X 0,Y 545.068,Z 277.587,A -85,B 0,C 180,E1 -3567.211,E2 -3567.211} C_VEL
LIN {X 0,Y 545.067,Z 277.59,A -85,B 0,C 180,E1 -3569.81,E2 -3569.81} C_VEL
LIN {X 0,Y 545.046,Z 277.587,A -85,B 0,C 180,E1 -3572.341,E2 -3572.341} C_VEL
LIN {X 0,Y 545.039,Z 277.586,A -85,B 0,C 180,E1 -3574.816,E2 -3574.816} C_VEL
LIN {X 0,Y 545.036,Z 277.589,A -85,B 0,C 180,E1 -3577.242,E2 -3577.242} C_VEL
LIN {X 0,Y 545.121,Z 277.578,A -85,B 0,C 180,E1 -3580.415,E2 -3580.415} C_VEL
LIN {X 0,Y 545.039,Z 277.59,A -85,B 0,C 180,E1 -3583.52,E2 -3583.52} C_VEL
LIN {X 0,Y 545.085,Z 277.588,A -85,B 0,C 180,E1 -3585.819,E2 -3585.819} C_VEL
LIN {X 0,Y 545.076,Z 277.582,A -85,B 0,C 180,E1 -3588.848,E2 -3588.848} C_VEL
LIN {X 0,Y 545.072,Z 277.588,A -85,B 0,C 180,E1 -3591.846,E2 -3591.846} C_VEL
LIN {X 0,Y 545.166,Z 277.572,A -85,B 0,C 180,E1 -3594.822,E2 -3594.822} C_VEL
LIN {X 0,Y 545.193,Z 277.57,A -85,B 0,C 180,E1 -3597.783,E2 -3597.783} C_VEL
LIN {X 0,Y 545.203,Z 277.569,A -85,B 0,C 180,E1 -3600.738,E2 -3600.738} C_VEL
LIN {X 0,Y 545.149,Z 277.574,A -85,B 0,C 180,E1 -3602.956,E2 -3602.956} C_VEL
LIN {X 0,Y 545.126,Z 277.578,A -85,B 0,C 180,E1 -3605.92,E2 -3605.92} C_VEL
LIN {X 0,Y 545.072,Z 277.586,A -85,B 0,C 180,E1 -3608.901,E2 -3608.901} C_VEL
LIN {X 0,Y 545.071,Z 277.584,A -85,B 0,C 180,E1 -3611.905,E2 -3611.905} C_VEL
LIN {X 0,Y 545.082,Z 277.586,A -85,B 0,C 180,E1 -3614.944,E2 -3614.944} C_VEL
LIN {X 0,Y 545.052,Z 277.586,A -85,B 0,C 180,E1 -3618.027,E2 -3618.027} C_VEL
LIN {X 0,Y 545.091,Z 277.584,A -85,B 0,C 180,E1 -3620.372,E2 -3620.372} C_VEL
LIN {X 0,Y 545.074,Z 277.582,A -85,B 0,C 180,E1 -3623.56,E2 -3623.56} C_VEL
LIN {X 0,Y 545.036,Z 277.587,A -85,B 0,C 180,E1 -3626.003,E2 -3626.003} C_VEL
LIN {X 0,Y 545.048,Z 277.592,A -85,B 0,C 180,E1 -3628.739,E2 -3628.739} C_VEL
LIN {X 0,Y 545.046,Z 277.585,A -85,B 0,C 180,E1 -3631.915,E2 -3631.915} C_VEL
LIN {X 0,Y 545.05,Z 277.588,A -85,B 0,C 180,E1 -3634.565,E2 -3634.565} C_VEL
LIN {X 0,Y 545.032,Z 277.594,A -85,B 0,C 180,E1 -3637.304,E2 -3637.304} C_VEL
LIN {X 0,Y 545.053,Z 277.584,A -85,B 0,C 180,E1 -3640.144,E2 -3640.144} C_VEL
LIN {X 0,Y 545.02,Z 277.597,A -85,B 0,C 180,E1 -3643.113,E2 -3643.113} C_VEL
LIN {X 0,Y 545.03,Z 277.587,A -85,B 0,C 180,E1 -3646.229,E2 -3646.229} C_VEL
LIN {X 0,Y 545.018,Z 277.592,A -85,B 0,C 180,E1 -3648.879,E2 -3648.879} C_VEL
LIN {X 0,Y 545.045,Z 277.59,A -85,B 0,C 180,E1 -3651.762,E2 -3651.762} C_VEL
LIN {X 0,Y 545.028,Z 277.588,A -85,B 0,C 180,E1 -3654.53,E2 -3654.53} C_VEL
LIN {X 0,Y 545.066,Z 277.588,A -85,B 0,C 180,E1 -3657.211,E2 -3657.211} C_VEL
LIN {X 0,Y 545.065,Z 277.591,A -85,B 0,C 180,E1 -3659.81,E2 -3659.81} C_VEL
LIN {X 0,Y 545.044,Z 277.588,A -85,B 0,C 180,E1 -3662.341,E2 -3662.341} C_VEL
LIN {X 0,Y 545.066,Z 277.661,A -85,B 0,C 180,E1 -3665.504,E2 -3665.504} C_VEL
LIN {X 0,Y 546.226,Z 284,A -85,B 0,C 180,E1 -3666.493,E2 -3666.493} C_VEL
LIN {X 0,Y 546.109,Z 298.942,A -85,B 0,C 180,E1 -3668.681,E2 -3668.681} C_VEL
LIN {X 0,Y 545.74,Z 320.628,A -85,B 0,C 180,E1 -3671.802,E2 -3671.802} C_VEL
LIN {X 0,Y 545.422,Z 343.591,A -85,B 0,C 180,E1 -3675.065,E2 -3675.065} C_VEL
LIN {X 0,Y 545.405,Z 346.132,A -85,B 0,C 180,E1 -3675.425,E2 -3675.425} C_VEL
LIN {X 0,Y 546.519,Z 354.717,A -85,B 0,C 180,E1 -3675.582,E2 -3675.582} C_VEL
LIN {X 0,Y 546.212,Z 454.76,A -85,B 0,C 180,E1 -3676.916,E2 -3676.916} C_VEL
LIN {X 0,Y 546.024,Z 468.068,A -85,B 0,C 180,E1 -3677.242,E2 -3677.242} C_VEL
LIN {X 0,Y 545.886,Z 480.265,A -85,B 0,C 180,E1 -3677.688,E2 -3677.688} C_VEL
LIN {X 0,Y 545.733,Z 492.612,A -85,B 0,C 180,E1 -3678.299,E2 -3678.299} C_VEL
LIN {X 0,Y 545.511,Z 504.185,A -85,B 0,C 180,E1 -3679.045,E2 -3679.045} C_VEL
LIN {X 0,Y 545.261,Z 514.599,A -85,B 0,C 180,E1 -3679.885,E2 -3679.885} C_VEL
LIN {X 0,Y 545.085,Z 523.109,A -85,B 0,C 180,E1 -3680.725,E2 -3680.725} C_VEL
LIN {X 0,Y 544.978,Z 530.957,A -85,B 0,C 180,E1 -3681.658,E2 -3681.658} C_VEL
LIN {X 0,Y 544.824,Z 538.618,A -85,B 0,C 180,E1 -3682.774,E2 -3682.774} C_VEL
LIN {X 0,Y 544.777,Z 545.677,A -85,B 0,C 180,E1 -3684.076,E2 -3684.076} C_VEL
LIN {X 0,Y 544.629,Z 550.371,A -85,B 0,C 180,E1 -3685.188,E2 -3685.188} C_VEL
LIN {X 0,Y 544.669,Z 553.957,A -85,B 0,C 180,E1 -3686.3,E2 -3686.3} C_VEL
LIN {X 0,Y 544.65,Z 555.806,A -85,B 0,C 180,E1 -3687.041,E2 -3687.041} C_VEL
LIN {X 0,Y 544.546,Z 558.182,A -85,B 0,C 180,E1 -3688.52,E2 -3688.52} C_VEL
LIN {X 0,Y 544.541,Z 559,A -85,B 0,C 180,E1 -3690,E2 -3690} C_VEL
LIN {X 0,Y 544.546,Z 558.184,A -85,B 0,C 180,E1 -3691.479,E2 -3691.479} C_VEL
LIN {X 0,Y 544.65,Z 555.811,A -85,B 0,C 180,E1 -3692.958,E2 -3692.958} C_VEL
LIN {X 0,Y 544.684,Z 552.897,A -85,B 0,C 180,E1 -3694.069,E2 -3694.069} C_VEL
LIN {X 0,Y 544.653,Z 548.95,A -85,B 0,C 180,E1 -3695.182,E2 -3695.182} C_VEL
LIN {X 0,Y 544.728,Z 543.648,A -85,B 0,C 180,E1 -3696.339,E2 -3696.339} C_VEL
LIN {X 0,Y 544.836,Z 537.469,A -85,B 0,C 180,E1 -3697.411,E2 -3697.411} C_VEL
LIN {X 0,Y 545.006,Z 529.481,A -85,B 0,C 180,E1 -3698.528,E2 -3698.528} C_VEL
LIN {X 0,Y 545.153,Z 521.337,A -85,B 0,C 180,E1 -3699.46,E2 -3699.46} C_VEL
LIN {X 0,Y 545.34,Z 511.402,A -85,B 0,C 180,E1 -3700.394,E2 -3700.394} C_VEL
LIN {X 0,Y 545.582,Z 500.55,A -85,B 0,C 180,E1 -3701.21,E2 -3701.21} C_VEL
LIN {X 0,Y 545.738,Z 489.121,A -85,B 0,C 180,E1 -3701.89,E2 -3701.89} C_VEL
LIN {X 0,Y 545.918,Z 476.875,A -85,B 0,C 180,E1 -3702.452,E2 -3702.452} C_VEL
LIN {X 0,Y 546.107,Z 464.043,A -85,B 0,C 180,E1 -3702.873,E2 -3702.873} C_VEL
LIN {X 0,Y 546.227,Z 450.45,A -85,B 0,C 180,E1 -3703.154,E2 -3703.154} C_VEL
LIN {X 0,Y 546.422,Z 353.196,A -85,B 0,C 180,E1 -3704.441,E2 -3704.441} C_VEL
LIN {X 0,Y 545.384,Z 346.19,A -85,B 0,C 180,E1 -3704.564,E2 -3704.564} C_VEL
LIN {X 0,Y 545.61,Z 324.764,A -85,B 0,C 180,E1 -3707.599,E2 -3707.599} C_VEL
LIN {X 0,Y 545.968,Z 305.619,A -85,B 0,C 180,E1 -3710.338,E2 -3710.338} C_VEL
LIN {X 0,Y 546.312,Z 285.185,A -85,B 0,C 180,E1 -3713.302,E2 -3713.302} C_VEL
LIN {X 0,Y 545.065,Z 277.593,A -85,B 0,C 180,E1 -3714.495,E2 -3714.495} C_VEL
LIN {X 0,Y 545.041,Z 277.591,A -85,B 0,C 180,E1 -3717.658,E2 -3717.658} C_VEL
LIN {X 0,Y 545.044,Z 277.598,A -85,B 0,C 180,E1 -3720.24,E2 -3720.24} C_VEL
LIN {X 0,Y 545.071,Z 277.587,A -85,B 0,C 180,E1 -3723.061,E2 -3723.061} C_VEL
LIN {X 0,Y 545.023,Z 277.592,A -85,B 0,C 180,E1 -3725.671,E2 -3725.671} C_VEL
LIN {X 0,Y 545.048,Z 277.594,A -85,B 0,C 180,E1 -3728.237,E2 -3728.237} C_VEL
LIN {X 0,Y 545.078,Z 277.583,A -85,B 0,C 180,E1 -3731.114,E2 -3731.114} C_VEL
LIN {X 0,Y 545.048,Z 277.591,A -85,B 0,C 180,E1 -3734.13,E2 -3734.13} C_VEL
LIN {X 0,Y 545.059,Z 277.585,A -85,B 0,C 180,E1 -3737.303,E2 -3737.303} C_VEL
LIN {X 0,Y 545.065,Z 277.584,A -85,B 0,C 180,E1 -3739.857,E2 -3739.857} C_VEL
LIN {X 0,Y 545.067,Z 277.586,A -85,B 0,C 180,E1 -3743.074,E2 -3743.074} C_VEL
LIN {X 0,Y 545.048,Z 277.59,A -85,B 0,C 180,E1 -3746.327,E2 -3746.327} C_VEL
LIN {X 0,Y 545.063,Z 277.588,A -85,B 0,C 180,E1 -3748.952,E2 -3748.952} C_VEL
LIN {X 0,Y 545.099,Z 277.578,A -85,B 0,C 180,E1 -3751.508,E2 -3751.508} C_VEL
LIN {X 0,Y 545.091,Z 277.587,A -85,B 0,C 180,E1 -3754.491,E2 -3754.491} C_VEL
LIN {X 0,Y 545.035,Z 277.589,A -85,B 0,C 180,E1 -3757.242,E2 -3757.242} C_VEL
LIN {X 0,Y 545.118,Z 277.58,A -85,B 0,C 180,E1 -3760.415,E2 -3760.415} C_VEL
LIN {X 0,Y 545.073,Z 277.582,A -85,B 0,C 180,E1 -3763.521,E2 -3763.521} C_VEL
LIN {X 0,Y 545.093,Z 277.58,A -85,B 0,C 180,E1 -3765.82,E2 -3765.82} C_VEL
LIN {X 0,Y 545.115,Z 277.587,A -85,B 0,C 180,E1 -3768.849,E2 -3768.849} C_VEL
LIN {X 0,Y 545.126,Z 277.574,A -85,B 0,C 180,E1 -3771.847,E2 -3771.847} C_VEL
LIN {X 0,Y 545.2,Z 277.576,A -85,B 0,C 180,E1 -3774.823,E2 -3774.823} C_VEL
LIN {X 0,Y 545.194,Z 277.567,A -85,B 0,C 180,E1 -3777.784,E2 -3777.784} C_VEL
LIN {X 0,Y 545.211,Z 277.571,A -85,B 0,C 180,E1 -3780.739,E2 -3780.739} C_VEL
LIN {X 0,Y 545.169,Z 277.581,A -85,B 0,C 180,E1 -3782.956,E2 -3782.956} C_VEL
LIN {X 0,Y 545.167,Z 277.57,A -85,B 0,C 180,E1 -3785.92,E2 -3785.92} C_VEL
LIN {X 0,Y 545.117,Z 277.585,A -85,B 0,C 180,E1 -3788.9,E2 -3788.9} C_VEL
LIN {X 0,Y 545.132,Z 277.575,A -85,B 0,C 180,E1 -3791.904,E2 -3791.904} C_VEL
LIN {X 0,Y 545.084,Z 277.588,A -85,B 0,C 180,E1 -3794.944,E2 -3794.944} C_VEL
LIN {X 0,Y 545.068,Z 277.582,A -85,B 0,C 180,E1 -3798.026,E2 -3798.026} C_VEL
LIN {X 0,Y 545.09,Z 277.581,A -85,B 0,C 180,E1 -3800.373,E2 -3800.373} C_VEL
LIN {X 0,Y 545.075,Z 277.586,A -85,B 0,C 180,E1 -3803.56,E2 -3803.56} C_VEL
LIN {X 0,Y 545.076,Z 277.582,A -85,B 0,C 180,E1 -3806.001,E2 -3806.001} C_VEL
LIN {X 0,Y 545.072,Z 277.585,A -85,B 0,C 180,E1 -3808.746,E2 -3808.746} C_VEL
LIN {X 0,Y 545.056,Z 277.587,A -85,B 0,C 180,E1 -3811.679,E2 -3811.679} C_VEL
LIN {X 0,Y 545.062,Z 277.585,A -85,B 0,C 180,E1 -3814.565,E2 -3814.565} C_VEL
LIN {X 0,Y 545.059,Z 277.589,A -85,B 0,C 180,E1 -3817.007,E2 -3817.007} C_VEL
LIN {X 0,Y 544.353,Z 277.682,A -85,B 0,C 180,E1 -3817.623,E2 -3817.623} C_VEL
LIN {X 0,Y 541.49,Z 278.038,A -85,B 0,C 180,E1 -3818.624,E2 -3818.624} C_VEL
LIN {X 0,Y 539.1,Z 278.335,A -85,B 0,C 180,E1 -3819.43,E2 -3819.43} C_VEL
LIN {X 0,Y 538.081,Z 278.455,A -85,B 0,C 180,E1 -3820.052,E2 -3820.052} C_VEL
LIN {X 0,Y 538.002,Z 278.463,A -85,B 0,C 180,E1 -3820.262,E2 -3820.262} C_VEL
LIN {X 0,Y 537.978,Z 278.471,A -85,B 0,C 180,E1 -3822.983,E2 -3822.983} C_VEL
LIN {X 0,Y 538.01,Z 278.465,A -85,B 0,C 180,E1 -3825.928,E2 -3825.928} C_VEL
LIN {X 0,Y 538.003,Z 278.471,A -85,B 0,C 180,E1 -3829.259,E2 -3829.259} C_VEL
LIN {X 0,Y 537.984,Z 278.468,A -85,B 0,C 180,E1 -3832.122,E2 -3832.122} C_VEL
LIN {X 0,Y 537.991,Z 278.466,A -85,B 0,C 180,E1 -3834.916,E2 -3834.916} C_VEL
LIN {X 0,Y 538.013,Z 278.472,A -85,B 0,C 180,E1 -3837.617,E2 -3837.617} C_VEL
LIN {X 0,Y 538.001,Z 278.468,A -85,B 0,C 180,E1 -3840.238,E2 -3840.238} C_VEL
LIN {X 0,Y 538.077,Z 278.491,A -85,B 0,C 180,E1 -3842.469,E2 -3842.469} C_VEL
LIN {X 0,Y 538.208,Z 284.773,A -85,B 0,C 180,E1 -3843.643,E2 -3843.643} C_VEL
LIN {X 0,Y 538.14,Z 298.688,A -85,B 0,C 180,E1 -3846.221,E2 -3846.221} C_VEL
LIN {X 0,Y 538.135,Z 299.07,A -85,B 0,C 180,E1 -3846.297,E2 -3846.297} C_VEL
LIN {X 0,Y 539.709,Z 308.096,A -85,B 0,C 180,E1 -3846.472,E2 -3846.472} C_VEL
LIN {X 0,Y 539.292,Z 405.811,A -85,B 0,C 180,E1 -3847.795,E2 -3847.795} C_VEL
LIN {X 0,Y 539.177,Z 419.456,A -85,B 0,C 180,E1 -3848.143,E2 -3848.143} C_VEL
LIN {X 0,Y 538.928,Z 432.407,A -85,B 0,C 180,E1 -3848.634,E2 -3848.634} C_VEL
LIN {X 0,Y 538.716,Z 444.64,A -85,B 0,C 180,E1 -3849.276,E2 -3849.276} C_VEL
LIN {X 0,Y 538.499,Z 455.415,A -85,B 0,C 180,E1 -3849.999,E2 -3849.999} C_VEL
LIN {X 0,Y 538.279,Z 465.639,A -85,B 0,C 180,E1 -3850.851,E2 -3850.851} C_VEL
LIN {X 0,Y 538.058,Z 474.267,A -85,B 0,C 180,E1 -3851.731,E2 -3851.731} C_VEL
LIN {X 0,Y 537.889,Z 482.505,A -85,B 0,C 180,E1 -3852.758,E2 -3852.758} C_VEL
LIN {X 0,Y 537.748,Z 489.801,A -85,B 0,C 180,E1 -3853.876,E2 -3853.876} C_VEL
LIN {X 0,Y 537.65,Z 496.506,A -85,B 0,C 180,E1 -3855.169,E2 -3855.169} C_VEL
LIN {X 0,Y 537.577,Z 501.338,A -85,B 0,C 180,E1 -3856.39,E2 -3856.39} C_VEL
LIN {X 0,Y 537.555,Z 503.722,A -85,B 0,C 180,E1 -3857.159,E2 -3857.159} C_VEL
LIN {X 0,Y 537.493,Z 505.663,A -85,B 0,C 180,E1 -3857.925,E2 -3857.925} C_VEL
LIN {X 0,Y 537.543,Z 507.155,A -85,B 0,C 180,E1 -3858.691,E2 -3858.691} C_VEL
LIN {X 0,Y 537.48,Z 508.836,A -85,B 0,C 180,E1 -3860.213,E2 -3860.213} C_VEL
LIN {X 0,Y 537.462,Z 509.092,A -85,B 0,C 180,E1 -3860.973,E2 -3860.973} C_VEL
LIN {X 0,Y 537.507,Z 508.926,A -85,B 0,C 180,E1 -3861.731,E2 -3861.731} C_VEL
LIN {X 0,Y 537.552,Z 507.382,A -85,B 0,C 180,E1 -3863.243,E2 -3863.243} C_VEL
LIN {X 0,Y 537.548,Z 506.03,A -85,B 0,C 180,E1 -3863.997,E2 -3863.997} C_VEL
LIN {X 0,Y 537.515,Z 503.178,A -85,B 0,C 180,E1 -3865.125,E2 -3865.125} C_VEL
LIN {X 0,Y 537.612,Z 499.304,A -85,B 0,C 180,E1 -3866.253,E2 -3866.253} C_VEL
LIN {X 0,Y 537.682,Z 494.326,A -85,B 0,C 180,E1 -3867.378,E2 -3867.378} C_VEL
LIN {X 0,Y 537.792,Z 488.083,A -85,B 0,C 180,E1 -3868.503,E2 -3868.503} C_VEL
LIN {X 0,Y 537.952,Z 480.289,A -85,B 0,C 180,E1 -3869.626,E2 -3869.626} C_VEL
LIN {X 0,Y 538.141,Z 470.627,A -85,B 0,C 180,E1 -3870.749,E2 -3870.749} C_VEL
LIN {X 0,Y 538.339,Z 460.575,A -85,B 0,C 180,E1 -3871.684,E2 -3871.684} C_VEL
LIN {X 0,Y 538.565,Z 449.249,A -85,B 0,C 180,E1 -3872.525,E2 -3872.525} C_VEL
LIN {X 0,Y 538.819,Z 438.113,A -85,B 0,C 180,E1 -3873.178,E2 -3873.178} C_VEL
LIN {X 0,Y 538.961,Z 426.814,A -85,B 0,C 180,E1 -3873.692,E2 -3873.692} C_VEL
LIN {X 0,Y 539.141,Z 413.866,A -85,B 0,C 180,E1 -3874.112,E2 -3874.112} C_VEL
LIN {X 0,Y 539.298,Z 401.415,A -85,B 0,C 180,E1 -3874.368,E2 -3874.368} C_VEL
LIN {X 0,Y 539.598,Z 306.961,A -85,B 0,C 180,E1 -3875.636,E2 -3875.636} C_VEL
LIN {X 0,Y 538.204,Z 299.153,A -85,B 0,C 180,E1 -3875.785,E2 -3875.785} C_VEL
LIN {X 0,Y 538.303,Z 284.085,A -85,B 0,C 180,E1 -3878.636,E2 -3878.636} C_VEL
LIN {X 0,Y 537.994,Z 278.471,A -85,B 0,C 180,E1 -3879.731,E2 -3879.731} C_VEL
LIN {X 0,Y 538.044,Z 278.463,A -85,B 0,C 180,E1 -3882.064,E2 -3882.064} C_VEL
LIN {X 0,Y 538.046,Z 278.46,A -85,B 0,C 180,E1 -3885.144,E2 -3885.144} C_VEL
LIN {X 0,Y 538.006,Z 278.466,A -85,B 0,C 180,E1 -3888.272,E2 -3888.272} C_VEL
LIN {X 0,Y 538.038,Z 278.467,A -85,B 0,C 180,E1 -3890.652,E2 -3890.652} C_VEL
LIN {X 0,Y 538.012,Z 278.462,A -85,B 0,C 180,E1 -3893.878,E2 -3893.878} C_VEL
LIN {X 0,Y 537.985,Z 278.467,A -85,B 0,C 180,E1 -3896.37,E2 -3896.37} C_VEL
LIN {X 0,Y 537.998,Z 278.473,A -85,B 0,C 180,E1 -3898.926,E2 -3898.926} C_VEL
LIN {X 0,Y 538.004,Z 278.463,A -85,B 0,C 180,E1 -3901.885,E2 -3901.885} C_VEL
LIN {X 0,Y 538.003,Z 278.466,A -85,B 0,C 180,E1 -3904.615,E2 -3904.615} C_VEL
LIN {X 0,Y 538.004,Z 278.473,A -85,B 0,C 180,E1 -3907.169,E2 -3907.169} C_VEL
LIN {X 0,Y 538.006,Z 278.464,A -85,B 0,C 180,E1 -3909.799,E2 -3909.799} C_VEL
LIN {X 0,Y 537.975,Z 278.472,A -85,B 0,C 180,E1 -3912.981,E2 -3912.981} C_VEL
LIN {X 0,Y 538.006,Z 278.464,A -85,B 0,C 180,E1 -3915.929,E2 -3915.929} C_VEL
LIN {X 0,Y 538.006,Z 278.47,A -85,B 0,C 180,E1 -3919.259,E2 -3919.259} C_VEL
LIN {X 0,Y 537.987,Z 278.466,A -85,B 0,C 180,E1 -3922.121,E2 -3922.121} C_VEL
LIN {X 0,Y 537.992,Z 278.466,A -85,B 0,C 180,E1 -3924.915,E2 -3924.915} C_VEL
LIN {X 0,Y 538.021,Z 278.471,A -85,B 0,C 180,E1 -3927.617,E2 -3927.617} C_VEL
LIN {X 0,Y 538.01,Z 278.464,A -85,B 0,C 180,E1 -3930.238,E2 -3930.238} C_VEL
LIN {X 0,Y 538.007,Z 278.462,A -85,B 0,C 180,E1 -3932.793,E2 -3932.793} C_VEL
LIN {X 0,Y 537.982,Z 278.468,A -85,B 0,C 180,E1 -3935.289,E2 -3935.289} C_VEL
LIN {X 0,Y 538.02,Z 278.467,A -85,B 0,C 180,E1 -3938.042,E2 -3938.042} C_VEL
LIN {X 0,Y 538.086,Z 278.458,A -85,B 0,C 180,E1 -3940.148,E2 -3940.148} C_VEL
LIN {X 0,Y 537.989,Z 278.466,A -85,B 0,C 180,E1 -3943.298,E2 -3943.298} C_VEL
LIN {X 0,Y 538.055,Z 278.461,A -85,B 0,C 180,E1 -3945.63,E2 -3945.63} C_VEL
LIN {X 0,Y 538.028,Z 278.461,A -85,B 0,C 180,E1 -3948.7,E2 -3948.7} C_VEL
LIN {X 0,Y 538.043,Z 278.462,A -85,B 0,C 180,E1 -3951.739,E2 -3951.739} C_VEL
LIN {X 0,Y 538.126,Z 278.449,A -85,B 0,C 180,E1 -3954.754,E2 -3954.754} C_VEL
LIN {X 0,Y 538.164,Z 278.446,A -85,B 0,C 180,E1 -3957.755,E2 -3957.755} C_VEL
LIN {X 0,Y 538.175,Z 278.445,A -85,B 0,C 180,E1 -3960.748,E2 -3960.748} C_VEL
LIN {X 0,Y 538.116,Z 278.45,A -85,B 0,C 180,E1 -3962.994,E2 -3962.994} C_VEL
LIN {X 0,Y 538.084,Z 278.456,A -85,B 0,C 180,E1 -3965.998,E2 -3965.998} C_VEL
LIN {X 0,Y 538.029,Z 278.462,A -85,B 0,C 180,E1 -3969.018,E2 -3969.018} C_VEL
LIN {X 0,Y 538.042,Z 278.461,A -85,B 0,C 180,E1 -3972.063,E2 -3972.063} C_VEL
LIN {X 0,Y 538.043,Z 278.46,A -85,B 0,C 180,E1 -3975.144,E2 -3975.144} C_VEL
LIN {X 0,Y 538.004,Z 278.466,A -85,B 0,C 180,E1 -3978.271,E2 -3978.271} C_VEL
LIN {X 0,Y 538.036,Z 278.468,A -85,B 0,C 180,E1 -3980.651,E2 -3980.651} C_VEL
LIN {X 0,Y 538.01,Z 278.462,A -85,B 0,C 180,E1 -3983.877,E2 -3983.877} C_VEL
LIN {X 0,Y 537.981,Z 278.468,A -85,B 0,C 180,E1 -3986.37,E2 -3986.37} C_VEL
LIN {X 0,Y 537.995,Z 278.474,A -85,B 0,C 180,E1 -3988.925,E2 -3988.925} C_VEL
LIN {X 0,Y 538.001,Z 278.463,A -85,B 0,C 180,E1 -3991.885,E2 -3991.885} C_VEL
LIN {X 0,Y 538.001,Z 278.467,A -85,B 0,C 180,E1 -3994.615,E2 -3994.615} C_VEL
LIN {X 0,Y 538.001,Z 278.472,A -85,B 0,C 180,E1 -3997.169,E2 -3997.169} C_VEL
LIN {X 0,Y 538.004,Z 278.464,A -85,B 0,C 180,E1 -3999.799,E2 -3999.799} C_VEL
LIN {X 0,Y 537.973,Z 278.473,A -85,B 0,C 180,E1 -4002.981,E2 -4002.981} C_VEL
LIN {X 0,Y 538.004,Z 278.464,A -85,B 0,C 180,E1 -4005.928,E2 -4005.928} C_VEL
LIN {X 0,Y 538.003,Z 278.471,A -85,B 0,C 180,E1 -4009.259,E2 -4009.259} C_VEL
LIN {X 0,Y 537.985,Z 278.466,A -85,B 0,C 180,E1 -4012.121,E2 -4012.121} C_VEL
LIN {X 0,Y 537.99,Z 278.466,A -85,B 0,C 180,E1 -4014.914,E2 -4014.914} C_VEL
LIN {X 0,Y 538.019,Z 278.471,A -85,B 0,C 180,E1 -4017.617,E2 -4017.617} C_VEL
LIN {X 0,Y 538.008,Z 278.465,A -85,B 0,C 180,E1 -4020.238,E2 -4020.238} C_VEL
LIN {X 0,Y 538.005,Z 278.465,A -85,B 0,C 180,E1 -4022.792,E2 -4022.792} C_VEL
LIN {X 0,Y 538.026,Z 278.528,A -85,B 0,C 180,E1 -4025.342,E2 -4025.342} C_VEL
LIN {X 0,Y 539.383,Z 286.41,A -85,B 0,C 180,E1 -4026.583,E2 -4026.583} C_VEL
LIN {X 0,Y 539.005,Z 306.409,A -85,B 0,C 180,E1 -4029.536,E2 -4029.536} C_VEL
LIN {X 0,Y 538.624,Z 325.24,A -85,B 0,C 180,E1 -4032.272,E2 -4032.272} C_VEL
LIN {X 0,Y 538.354,Z 345.895,A -85,B 0,C 180,E1 -4035.243,E2 -4035.243} C_VEL
LIN {X 0,Y 539.636,Z 355.665,A -85,B 0,C 180,E1 -4035.411,E2 -4035.411} C_VEL
LIN {X 0,Y 539.291,Z 454.413,A -85,B 0,C 180,E1 -4036.745,E2 -4036.745} C_VEL
LIN {X 0,Y 539.107,Z 467.729,A -85,B 0,C 180,E1 -4037.076,E2 -4037.076} C_VEL
LIN {X 0,Y 538.928,Z 479.927,A -85,B 0,C 180,E1 -4037.526,E2 -4037.526} C_VEL
LIN {X 0,Y 538.767,Z 491.401,A -85,B 0,C 180,E1 -4038.095,E2 -4038.095} C_VEL
LIN {X 0,Y 538.536,Z 502.573,A -85,B 0,C 180,E1 -4038.806,E2 -4038.806} C_VEL
LIN {X 0,Y 538.261,Z 513.268,A -85,B 0,C 180,E1 -4039.657,E2 -4039.657} C_VEL
LIN {X 0,Y 538.068,Z 522.911,A -85,B 0,C 180,E1 -4040.603,E2 -4040.603} C_VEL
LIN {X 0,Y 537.921,Z 530.819,A -85,B 0,C 180,E1 -4041.547,E2 -4041.547} C_VEL
LIN {X 0,Y 537.755,Z 538.542,A -85,B 0,C 180,E1 -4042.679,E2 -4042.679} C_VEL
LIN {X 0,Y 537.693,Z 545.664,A -85,B 0,C 180,E1 -4043.997,E2 -4043.997} C_VEL
LIN {X 0,Y 537.54,Z 550.371,A -85,B 0,C 180,E1 -4045.124,E2 -4045.124} C_VEL
LIN {X 0,Y 537.591,Z 553.956,A -85,B 0,C 180,E1 -4046.252,E2 -4046.252} C_VEL
LIN {X 0,Y 537.551,Z 555.805,A -85,B 0,C 180,E1 -4047.002,E2 -4047.002} C_VEL
LIN {X 0,Y 537.451,Z 558.181,A -85,B 0,C 180,E1 -4048.501,E2 -4048.501} C_VEL
LIN {X 0,Y 537.442,Z 559,A -85,B 0,C 180,E1 -4050,E2 -4050} C_VEL
LIN {X 0,Y 537.451,Z 558.184,A -85,B 0,C 180,E1 -4051.498,E2 -4051.498} C_VEL
LIN {X 0,Y 537.551,Z 555.811,A -85,B 0,C 180,E1 -4052.997,E2 -4052.997} C_VEL
LIN {X 0,Y 537.603,Z 552.896,A -85,B 0,C 180,E1 -4054.123,E2 -4054.123} C_VEL
LIN {X 0,Y 537.587,Z 548.949,A -85,B 0,C 180,E1 -4055.25,E2 -4055.25} C_VEL
LIN {X 0,Y 537.642,Z 544.101,A -85,B 0,C 180,E1 -4056.325,E2 -4056.325} C_VEL
LIN {X 0,Y 537.771,Z 537.382,A -85,B 0,C 180,E1 -4057.509,E2 -4057.509} C_VEL
LIN {X 0,Y 537.953,Z 529.329,A -85,B 0,C 180,E1 -4058.64,E2 -4058.64} C_VEL
LIN {X 0,Y 538.115,Z 521.124,A -85,B 0,C 180,E1 -4059.585,E2 -4059.585} C_VEL
LIN {X 0,Y 538.338,Z 511.122,A -85,B 0,C 180,E1 -4060.531,E2 -4060.531} C_VEL
LIN {X 0,Y 538.549,Z 501.26,A -85,B 0,C 180,E1 -4061.288,E2 -4061.288} C_VEL
LIN {X 0,Y 538.736,Z 490.05,A -85,B 0,C 180,E1 -4061.979,E2 -4061.979} C_VEL
LIN {X 0,Y 538.94,Z 477.66,A -85,B 0,C 180,E1 -4062.568,E2 -4062.568} C_VEL
LIN {X 0,Y 539.151,Z 464.604,A -85,B 0,C 180,E1 -4063.018,E2 -4063.018} C_VEL
LIN {X 0,Y 539.314,Z 451.592,A -85,B 0,C 180,E1 -4063.302,E2 -4063.302} C_VEL
LIN {X 0,Y 539.589,Z 354.33,A -85,B 0,C 180,E1 -4064.608,E2 -4064.608} C_VEL
LIN {X 0,Y 538.361,Z 345.745,A -85,B 0,C 180,E1 -4064.773,E2 -4064.773} C_VEL
LIN {X 0,Y 538.65,Z 323.788,A -85,B 0,C 180,E1 -4067.925,E2 -4067.925} C_VEL
LIN {X 0,Y 539.033,Z 303.905,A -85,B 0,C 180,E1 -4070.811,E2 -4070.811} C_VEL
LIN {X 0,Y 539.35,Z 286.19,A -85,B 0,C 180,E1 -4073.417,E2 -4073.417} C_VEL
LIN {X 0,Y 538.024,Z 278.469,A -85,B 0,C 180,E1 -4074.662,E2 -4074.662} C_VEL
LIN {X 0,Y 538.009,Z 278.472,A -85,B 0,C 180,E1 -4078.051,E2 -4078.051} C_VEL
LIN {X 0,Y 538.006,Z 278.472,A -85,B 0,C 180,E1 -4080.627,E2 -4080.627} C_VEL
LIN {X 0,Y 538.018,Z 278.465,A -85,B 0,C 180,E1 -4083.278,E2 -4083.278} C_VEL
LIN {X 0,Y 537.988,Z 278.471,A -85,B 0,C 180,E1 -4086.004,E2 -4086.004} C_VEL
LIN {X 0,Y 538.009,Z 278.466,A -85,B 0,C 180,E1 -4088.83,E2 -4088.83} C_VEL
LIN {X 0,Y 538.028,Z 278.461,A -85,B 0,C 180,E1 -4091.773,E2 -4091.773} C_VEL
LIN {X 0,Y 538.004,Z 278.467,A -85,B 0,C 180,E1 -4094.862,E2 -4094.862} C_VEL
LIN {X 0,Y 538.016,Z 278.463,A -85,B 0,C 180,E1 -4097.214,E2 -4097.214} C_VEL
LIN {X 0,Y 538.022,Z 278.465,A -85,B 0,C 180,E1 -4100.203,E2 -4100.203} C_VEL
LIN {X 0,Y 538.021,Z 278.463,A -85,B 0,C 180,E1 -4103.067,E2 -4103.067} C_VEL
LIN {X 0,Y 538.009,Z 278.462,A -85,B 0,C 180,E1 -4105.826,E2 -4105.826} C_VEL
LIN {X 0,Y 538.006,Z 278.471,A -85,B 0,C 180,E1 -4108.498,E2 -4108.498} C_VEL
LIN {X 0,Y 538.039,Z 278.46,A -85,B 0,C 180,E1 -4111.099,E2 -4111.099} C_VEL
LIN {X 0,Y 538.038,Z 278.459,A -85,B 0,C 180,E1 -4113.633,E2 -4113.633} C_VEL
LIN {X 0,Y 538.003,Z 278.463,A -85,B 0,C 180,E1 -4116.122,E2 -4116.122} C_VEL
LIN {X 0,Y 538.037,Z 278.458,A -85,B 0,C 180,E1 -4119.349,E2 -4119.349} C_VEL
LIN {X 0,Y 538.051,Z 278.464,A -85,B 0,C 180,E1 -4122.517,E2 -4122.517} C_VEL
LIN {X 0,Y 538.062,Z 278.456,A -85,B 0,C 180,E1 -4125.631,E2 -4125.631} C_VEL
LIN {X 0,Y 538.074,Z 278.461,A -85,B 0,C 180,E1 -4128.702,E2 -4128.702} C_VEL
LIN {X 0,Y 538.083,Z 278.452,A -85,B 0,C 180,E1 -4131.74,E2 -4131.74} C_VEL
LIN {X 0,Y 538.157,Z 278.452,A -85,B 0,C 180,E1 -4134.755,E2 -4134.755} C_VEL
LIN {X 0,Y 538.166,Z 278.443,A -85,B 0,C 180,E1 -4137.755,E2 -4137.755} C_VEL
LIN {X 0,Y 538.181,Z 278.447,A -85,B 0,C 180,E1 -4140.748,E2 -4140.748} C_VEL
LIN {X 0,Y 538.135,Z 278.456,A -85,B 0,C 180,E1 -4142.995,E2 -4142.995} C_VEL
LIN {X 0,Y 538.12,Z 278.448,A -85,B 0,C 180,E1 -4145.998,E2 -4145.998} C_VEL
LIN {X 0,Y 538.068,Z 278.463,A -85,B 0,C 180,E1 -4149.018,E2 -4149.018} C_VEL
LIN {X 0,Y 538.081,Z 278.453,A -85,B 0,C 180,E1 -4152.063,E2 -4152.063} C_VEL
LIN {X 0,Y 538.043,Z 278.467,A -85,B 0,C 180,E1 -4155.144,E2 -4155.144} C_VEL
LIN {X 0,Y 538.022,Z 278.46,A -85,B 0,C 180,E1 -4158.271,E2 -4158.271} C_VEL
LIN {X 0,Y 538.036,Z 278.462,A -85,B 0,C 180,E1 -4160.652,E2 -4160.652} C_VEL
LIN {X 0,Y 537.998,Z 278.465,A -85,B 0,C 180,E1 -4163.889,E2 -4163.889} C_VEL
LIN {X 0,Y 538.038,Z 278.459,A -85,B 0,C 180,E1 -4166.367,E2 -4166.367} C_VEL
LIN {X 0,Y 538.028,Z 278.465,A -85,B 0,C 180,E1 -4168.934,E2 -4168.934} C_VEL
LIN {X 0,Y 538.008,Z 278.463,A -85,B 0,C 180,E1 -4171.888,E2 -4171.888} C_VEL
LIN {X 0,Y 538.012,Z 278.463,A -85,B 0,C 180,E1 -4174.618,E2 -4174.618} C_VEL
LIN {X 0,Y 538.003,Z 278.471,A -85,B 0,C 180,E1 -4177.17,E2 -4177.17} C_VEL
LIN {X 0,Y 538.019,Z 278.464,A -85,B 0,C 180,E1 -4179.798,E2 -4179.798} C_VEL
LIN {X 0,Y 538.002,Z 278.463,A -85,B 0,C 180,E1 -4180.262,E2 -4180.262} C_VEL
LIN {X 0,Y 537.341,Z 278.549,A -85,B 0,C 180,E1 -4180.888,E2 -4180.888} C_VEL
LIN {X 0,Y 534.484,Z 278.912,A -85,B 0,C 180,E1 -4181.902,E2 -4181.902} C_VEL
LIN {X 0,Y 532.063,Z 279.217,A -85,B 0,C 180,E1 -4182.719,E2 -4182.719} C_VEL
LIN {X 0,Y 531.02,Z 279.344,A -85,B 0,C 180,E1 -4183.35,E2 -4183.35} C_VEL
LIN {X 0,Y 530.934,Z 279.351,A -85,B 0,C 180,E1 -4183.564,E2 -4183.564} C_VEL
LIN {X 0,Y 530.937,Z 279.344,A -85,B 0,C 180,E1 -4186.503,E2 -4186.503} C_VEL
LIN {X 0,Y 530.948,Z 279.351,A -85,B 0,C 180,E1 -4189.565,E2 -4189.565} C_VEL
LIN {X 0,Y 530.938,Z 279.344,A -85,B 0,C 180,E1 -4192.582,E2 -4192.582} C_VEL
LIN {X 0,Y 530.977,Z 279.344,A -85,B 0,C 180,E1 -4195.31,E2 -4195.31} C_VEL
LIN {X 0,Y 530.959,Z 279.346,A -85,B 0,C 180,E1 -4198.032,E2 -4198.032} C_VEL
LIN {X 0,Y 530.965,Z 279.345,A -85,B 0,C 180,E1 -4200.88,E2 -4200.88} C_VEL
LIN {X 0,Y 531.019,Z 279.397,A -85,B 0,C 180,E1 -4202.405,E2 -4202.405} C_VEL
LIN {X 0,Y 531.225,Z 285.2,A -85,B 0,C 180,E1 -4203.481,E2 -4203.481} C_VEL
LIN {X 0,Y 531.132,Z 299.226,A -85,B 0,C 180,E1 -4206.092,E2 -4206.092} C_VEL
LIN {X 0,Y 532.864,Z 309.414,A -85,B 0,C 180,E1 -4206.295,E2 -4206.295} C_VEL
LIN {X 0,Y 532.407,Z 405.763,A -85,B 0,C 180,E1 -4207.613,E2 -4207.613} C_VEL
LIN {X 0,Y 532.294,Z 419.259,A -85,B 0,C 180,E1 -4207.957,E2 -4207.957} C_VEL
LIN {X 0,Y 532.031,Z 432.163,A -85,B 0,C 180,E1 -4208.445,E2 -4208.445} C_VEL
LIN {X 0,Y 531.79,Z 444.548,A -85,B 0,C 180,E1 -4209.095,E2 -4209.095} C_VEL
LIN {X 0,Y 531.519,Z 456.284,A -85,B 0,C 180,E1 -4209.893,E2 -4209.893} C_VEL
LIN {X 0,Y 531.297,Z 466.738,A -85,B 0,C 180,E1 -4210.79,E2 -4210.79} C_VEL
LIN {X 0,Y 531.008,Z 476.893,A -85,B 0,C 180,E1 -4211.879,E2 -4211.879} C_VEL
LIN {X 0,Y 530.829,Z 484.561,A -85,B 0,C 180,E1 -4212.893,E2 -4212.893} C_VEL
LIN {X 0,Y 530.656,Z 491.678,A -85,B 0,C 180,E1 -4214.05,E2 -4214.05} C_VEL
LIN {X 0,Y 530.588,Z 497.419,A -85,B 0,C 180,E1 -4215.227,E2 -4215.227} C_VEL
LIN {X 0,Y 530.5,Z 502.533,A -85,B 0,C 180,E1 -4216.595,E2 -4216.595} C_VEL
LIN {X 0,Y 530.413,Z 505.711,A -85,B 0,C 180,E1 -4217.761,E2 -4217.761} C_VEL
LIN {X 0,Y 530.451,Z 507.472,A -85,B 0,C 180,E1 -4218.65,E2 -4218.65} C_VEL
LIN {X 0,Y 530.39,Z 509.091,A -85,B 0,C 180,E1 -4220.081,E2 -4220.081} C_VEL
LIN {X 0,Y 530.417,Z 509.314,A -85,B 0,C 180,E1 -4221.62,E2 -4221.62} C_VEL
LIN {X 0,Y 530.428,Z 508.802,A -85,B 0,C 180,E1 -4222.387,E2 -4222.387} C_VEL
LIN {X 0,Y 530.478,Z 507.303,A -85,B 0,C 180,E1 -4223.536,E2 -4223.536} C_VEL
LIN {X 0,Y 530.436,Z 503.836,A -85,B 0,C 180,E1 -4225.06,E2 -4225.06} C_VEL
LIN {X 0,Y 530.534,Z 500.074,A -85,B 0,C 180,E1 -4226.203,E2 -4226.203} C_VEL
LIN {X 0,Y 530.621,Z 495.213,A -85,B 0,C 180,E1 -4227.343,E2 -4227.343} C_VEL
LIN {X 0,Y 530.721,Z 489.115,A -85,B 0,C 180,E1 -4228.483,E2 -4228.483} C_VEL
LIN {X 0,Y 530.917,Z 481.531,A -85,B 0,C 180,E1 -4229.621,E2 -4229.621} C_VEL
LIN {X 0,Y 531.12,Z 472.05,A -85,B 0,C 180,E1 -4230.759,E2 -4230.759} C_VEL
LIN {X 0,Y 531.362,Z 462.288,A -85,B 0,C 180,E1 -4231.706,E2 -4231.706} C_VEL
LIN {X 0,Y 531.57,Z 451.328,A -85,B 0,C 180,E1 -4232.558,E2 -4232.558} C_VEL
LIN {X 0,Y 531.815,Z 440.615,A -85,B 0,C 180,E1 -4233.22,E2 -4233.22} C_VEL
LIN {X 0,Y 532.031,Z 427.727,A -85,B 0,C 180,E1 -4233.835,E2 -4233.835} C_VEL
LIN {X 0,Y 532.228,Z 415.093,A -85,B 0,C 180,E1 -4234.26,E2 -4234.26} C_VEL
LIN {X 0,Y 532.41,Z 401.739,A -85,B 0,C 180,E1 -4234.543,E2 -4234.543} C_VEL
LIN {X 0,Y 532.747,Z 307.753,A -85,B 0,C 180,E1 -4235.821,E2 -4235.821} C_VEL
LIN {X 0,Y 531.192,Z 299.281,A -85,B 0,C 180,E1 -4236.005,E2 -4236.005} C_VEL
LIN {X 0,Y 531.305,Z 284.77,A -85,B 0,C 180,E1 -4238.75,E2 -4238.75} C_VEL
LIN {X 0,Y 530.947,Z 279.35,A -85,B 0,C 180,E1 -4239.813,E2 -4239.813} C_VEL
LIN {X 0,Y 531.015,Z 279.34,A -85,B 0,C 180,E1 -4242.226,E2 -4242.226} C_VEL
LIN {X 0,Y 530.991,Z 279.337,A -85,B 0,C 180,E1 -4245.35,E2 -4245.35} C_VEL
LIN {X 0,Y 530.964,Z 279.346,A -85,B 0,C 180,E1 -4248.523,E2 -4248.523} C_VEL
LIN {X 0,Y 531.001,Z 279.343,A -85,B 0,C 180,E1 -4250.938,E2 -4250.938} C_VEL
LIN {X 0,Y 530.955,Z 279.342,A -85,B 0,C 180,E1 -4254.226,E2 -4254.226} C_VEL
LIN {X 0,Y 530.95,Z 279.349,A -85,B 0,C 180,E1 -4256.747,E2 -4256.747} C_VEL
LIN {X 0,Y 530.96,Z 279.344,A -85,B 0,C 180,E1 -4259.324,E2 -4259.324} C_VEL
LIN {X 0,Y 530.961,Z 279.34,A -85,B 0,C 180,E1 -4262.098,E2 -4262.098} C_VEL
LIN {X 0,Y 530.964,Z 279.346,A -85,B 0,C 180,E1 -4264.849,E2 -4264.849} C_VEL
LIN {X 0,Y 530.968,Z 279.343,A -85,B 0,C 180,E1 -4267.508,E2 -4267.508} C_VEL
LIN {X 0,Y 530.946,Z 279.342,A -85,B 0,C 180,E1 -4270.437,E2 -4270.437} C_VEL
LIN {X 0,Y 530.932,Z 279.35,A -85,B 0,C 180,E1 -4273.499,E2 -4273.499} C_VEL
LIN {X 0,Y 530.97,Z 279.344,A -85,B 0,C 180,E1 -4275.623,E2 -4275.623} C_VEL
LIN {X 0,Y 530.94,Z 279.346,A -85,B 0,C 180,E1 -4278.983,E2 -4278.983} C_VEL
LIN {X 0,Y 530.953,Z 279.35,A -85,B 0,C 180,E1 -4281.528,E2 -4281.528} C_VEL
LIN {X 0,Y 530.952,Z 279.341,A -85,B 0,C 180,E1 -4284.379,E2 -4284.379} C_VEL
LIN {X 0,Y 530.972,Z 279.342,A -85,B 0,C 180,E1 -4287.133,E2 -4287.133} C_VEL
LIN {X 0,Y 530.957,Z 279.348,A -85,B 0,C 180,E1 -4289.802,E2 -4289.802} C_VEL
LIN {X 0,Y 530.967,Z 279.34,A -85,B 0,C 180,E1 -4292.478,E2 -4292.478} C_VEL
LIN {X 0,Y 530.948,Z 279.342,A -85,B 0,C 180,E1 -4294.939,E2 -4294.939} C_VEL
LIN {X 0,Y 530.982,Z 279.346,A -85,B 0,C 180,E1 -4297.898,E2 -4297.898} C_VEL
LIN {X 0,Y 530.984,Z 279.338,A -85,B 0,C 180,E1 -4300.677,E2 -4300.677} C_VEL
LIN {X 0,Y 530.957,Z 279.341,A -85,B 0,C 180,E1 -4303.07,E2 -4303.07} C_VEL
LIN {X 0,Y 531.012,Z 279.336,A -85,B 0,C 180,E1 -4305.435,E2 -4305.435} C_VEL
LIN {X 0,Y 530.99,Z 279.339,A -85,B 0,C 180,E1 -4308.548,E2 -4308.548} C_VEL
LIN {X 0,Y 530.993,Z 279.339,A -85,B 0,C 180,E1 -4311.628,E2 -4311.628} C_VEL
LIN {X 0,Y 531.088,Z 279.327,A -85,B 0,C 180,E1 -4314.685,E2 -4314.685} C_VEL
LIN {X 0,Y 531.136,Z 279.321,A -85,B 0,C 180,E1 -4317.725,E2 -4317.725} C_VEL
LIN {X 0,Y 531.125,Z 279.323,A -85,B 0,C 180,E1 -4320.758,E2 -4320.758} C_VEL
LIN {X 0,Y 531.057,Z 279.329,A -85,B 0,C 180,E1 -4323.034,E2 -4323.034} C_VEL
LIN {X 0,Y 531.045,Z 279.334,A -85,B 0,C 180,E1 -4326.077,E2 -4326.077} C_VEL
LIN {X 0,Y 530.994,Z 279.337,A -85,B 0,C 180,E1 -4329.139,E2 -4329.139} C_VEL
LIN {X 0,Y 531.012,Z 279.338,A -85,B 0,C 180,E1 -4332.225,E2 -4332.225} C_VEL
LIN {X 0,Y 530.989,Z 279.337,A -85,B 0,C 180,E1 -4335.35,E2 -4335.35} C_VEL
LIN {X 0,Y 530.961,Z 279.347,A -85,B 0,C 180,E1 -4338.522,E2 -4338.522} C_VEL
LIN {X 0,Y 530.998,Z 279.342,A -85,B 0,C 180,E1 -4340.938,E2 -4340.938} C_VEL
LIN {X 0,Y 530.952,Z 279.343,A -85,B 0,C 180,E1 -4344.226,E2 -4344.226} C_VEL
LIN {X 0,Y 530.947,Z 279.35,A -85,B 0,C 180,E1 -4346.747,E2 -4346.747} C_VEL
LIN {X 0,Y 530.958,Z 279.344,A -85,B 0,C 180,E1 -4349.324,E2 -4349.324} C_VEL
LIN {X 0,Y 530.959,Z 279.34,A -85,B 0,C 180,E1 -4352.098,E2 -4352.098} C_VEL
LIN {X 0,Y 530.961,Z 279.347,A -85,B 0,C 180,E1 -4354.849,E2 -4354.849} C_VEL
LIN {X 0,Y 530.966,Z 279.343,A -85,B 0,C 180,E1 -4357.508,E2 -4357.508} C_VEL
LIN {X 0,Y 530.944,Z 279.343,A -85,B 0,C 180,E1 -4360.436,E2 -4360.436} C_VEL
LIN {X 0,Y 530.929,Z 279.35,A -85,B 0,C 180,E1 -4363.498,E2 -4363.498} C_VEL
LIN {X 0,Y 530.968,Z 279.344,A -85,B 0,C 180,E1 -4365.623,E2 -4365.623} C_VEL
LIN {X 0,Y 530.937,Z 279.347,A -85,B 0,C 180,E1 -4368.982,E2 -4368.982} C_VEL
LIN {X 0,Y 530.95,Z 279.35,A -85,B 0,C 180,E1 -4371.528,E2 -4371.528} C_VEL
LIN {X 0,Y 530.95,Z 279.342,A -85,B 0,C 180,E1 -4374.379,E2 -4374.379} C_VEL
LIN {X 0,Y 530.969,Z 279.343,A -85,B 0,C 180,E1 -4377.133,E2 -4377.133} C_VEL
LIN {X 0,Y 530.955,Z 279.349,A -85,B 0,C 180,E1 -4379.802,E2 -4379.802} C_VEL
LIN {X 0,Y 530.965,Z 279.342,A -85,B 0,C 180,E1 -4382.478,E2 -4382.478} C_VEL
LIN {X 0,Y 530.996,Z 279.396,A -85,B 0,C 180,E1 -4385.177,E2 -4385.177} C_VEL
LIN {X 0,Y 532.426,Z 287.453,A -85,B 0,C 180,E1 -4386.465,E2 -4386.465} C_VEL
LIN {X 0,Y 532.036,Z 307.744,A -85,B 0,C 180,E1 -4389.503,E2 -4389.503} C_VEL
LIN {X 0,Y 531.607,Z 328.077,A -85,B 0,C 180,E1 -4392.496,E2 -4392.496} C_VEL
LIN {X 0,Y 531.332,Z 345.509,A -85,B 0,C 180,E1 -4395.036,E2 -4395.036} C_VEL
LIN {X 0,Y 532.776,Z 356.41,A -85,B 0,C 180,E1 -4395.234,E2 -4395.234} C_VEL
LIN {X 0,Y 532.382,Z 454.067,A -85,B 0,C 180,E1 -4396.57,E2 -4396.57} C_VEL
LIN {X 0,Y 532.159,Z 467.388,A -85,B 0,C 180,E1 -4396.904,E2 -4396.904} C_VEL
LIN {X 0,Y 531.966,Z 479.589,A -85,B 0,C 180,E1 -4397.36,E2 -4397.36} C_VEL
LIN {X 0,Y 531.76,Z 491.584,A -85,B 0,C 180,E1 -4397.966,E2 -4397.966} C_VEL
LIN {X 0,Y 531.5,Z 503.537,A -85,B 0,C 180,E1 -4398.753,E2 -4398.753} C_VEL
LIN {X 0,Y 531.209,Z 514.01,A -85,B 0,C 180,E1 -4399.615,E2 -4399.615} C_VEL
LIN {X 0,Y 531.019,Z 522.579,A -85,B 0,C 180,E1 -4400.477,E2 -4400.477} C_VEL
LIN {X 0,Y 530.86,Z 530.487,A -85,B 0,C 180,E1 -4401.434,E2 -4401.434} C_VEL
LIN {X 0,Y 530.675,Z 538.211,A -85,B 0,C 180,E1 -4402.581,E2 -4402.581} C_VEL
LIN {X 0,Y 530.585,Z 545.335,A -85,B 0,C 180,E1 -4403.917,E2 -4403.917} C_VEL
LIN {X 0,Y 530.459,Z 550.071,A -85,B 0,C 180,E1 -4405.059,E2 -4405.059} C_VEL
LIN {X 0,Y 530.516,Z 553.697,A -85,B 0,C 180,E1 -4406.202,E2 -4406.202} C_VEL
LIN {X 0,Y 530.457,Z 555.563,A -85,B 0,C 180,E1 -4406.962,E2 -4406.962} C_VEL
LIN {X 0,Y 530.41,Z 556.963,A -85,B 0,C 180,E1 -4407.721,E2 -4407.721} C_VEL
LIN {X 0,Y 530.345,Z 558.57,A -85,B 0,C 180,E1 -4409.24,E2 -4409.24} C_VEL
LIN {X 0,Y 530.346,Z 558.788,A -85,B 0,C 180,E1 -4410,E2 -4410} C_VEL
LIN {X 0,Y 530.361,Z 557.962,A -85,B 0,C 180,E1 -4411.518,E2 -4411.518} C_VEL
LIN {X 0,Y 530.41,Z 556.966,A -85,B 0,C 180,E1 -4412.278,E2 -4412.278} C_VEL
LIN {X 0,Y 530.457,Z 555.567,A -85,B 0,C 180,E1 -4413.037,E2 -4413.037} C_VEL
LIN {X 0,Y 530.522,Z 552.623,A -85,B 0,C 180,E1 -4414.178,E2 -4414.178} C_VEL
LIN {X 0,Y 530.524,Z 548.634,A -85,B 0,C 180,E1 -4415.32,E2 -4415.32} C_VEL
LIN {X 0,Y 530.594,Z 542.914,A -85,B 0,C 180,E1 -4416.578,E2 -4416.578} C_VEL
LIN {X 0,Y 530.719,Z 535.802,A -85,B 0,C 180,E1 -4417.801,E2 -4417.801} C_VEL
LIN {X 0,Y 530.914,Z 527.492,A -85,B 0,C 180,E1 -4418.948,E2 -4418.948} C_VEL
LIN {X 0,Y 531.101,Z 518.976,A -85,B 0,C 180,E1 -4419.905,E2 -4419.905} C_VEL
LIN {X 0,Y 531.354,Z 508.458,A -85,B 0,C 180,E1 -4420.864,E2 -4420.864} C_VEL
LIN {X 0,Y 531.635,Z 497.47,A -85,B 0,C 180,E1 -4421.67,E2 -4421.67} C_VEL
LIN {X 0,Y 531.861,Z 486.657,A -85,B 0,C 180,E1 -4422.302,E2 -4422.302} C_VEL
LIN {X 0,Y 532.031,Z 474.964,A -85,B 0,C 180,E1 -4422.831,E2 -4422.831} C_VEL
LIN {X 0,Y 532.317,Z 461.505,A -85,B 0,C 180,E1 -4423.261,E2 -4423.261} C_VEL
LIN {X 0,Y 532.435,Z 449.724,A -85,B 0,C 180,E1 -4423.501,E2 -4423.501} C_VEL
LIN {X 0,Y 532.646,Z 354.321,A -85,B 0,C 180,E1 -4424.798,E2 -4424.798} C_VEL
LIN {X 0,Y 531.328,Z 345.404,A -85,B 0,C 180,E1 -4424.973,E2 -4424.973} C_VEL
LIN {X 0,Y 531.71,Z 322.52,A -85,B 0,C 180,E1 -4428.302,E2 -4428.302} C_VEL
LIN {X 0,Y 532.048,Z 303.55,A -85,B 0,C 180,E1 -4431.097,E2 -4431.097} C_VEL
LIN {X 0,Y 532.386,Z 287.195,A -85,B 0,C 180,E1 -4433.536,E2 -4433.536} C_VEL
LIN {X 0,Y 531.012,Z 279.341,A -85,B 0,C 180,E1 -4434.795,E2 -4434.795} C_VEL
LIN {X 0,Y 530.961,Z 279.345,A -85,B 0,C 180,E1 -4437.598,E2 -4437.598} C_VEL
LIN {X 0,Y 530.952,Z 279.354,A -85,B 0,C 180,E1 -4440.197,E2 -4440.197} C_VEL
LIN {X 0,Y 530.965,Z 279.346,A -85,B 0,C 180,E1 -4442.866,E2 -4442.866} C_VEL
LIN {X 0,Y 530.948,Z 279.345,A -85,B 0,C 180,E1 -4445.62,E2 -4445.62} C_VEL
LIN {X 0,Y 530.962,Z 279.346,A -85,B 0,C 180,E1 -4448.653,E2 -4448.653} C_VEL
LIN {X 0,Y 530.991,Z 279.336,A -85,B 0,C 180,E1 -4451.435,E2 -4451.435} C_VEL
LIN {X 0,Y 530.972,Z 279.348,A -85,B 0,C 180,E1 -4454.548,E2 -4454.548} C_VEL
LIN {X 0,Y 530.979,Z 279.34,A -85,B 0,C 180,E1 -4457.834,E2 -4457.834} C_VEL
LIN {X 0,Y 530.985,Z 279.347,A -85,B 0,C 180,E1 -4460.556,E2 -4460.556} C_VEL
LIN {X 0,Y 530.952,Z 279.342,A -85,B 0,C 180,E1 -4463.441,E2 -4463.441} C_VEL
LIN {X 0,Y 530.953,Z 279.344,A -85,B 0,C 180,E1 -4466.225,E2 -4466.225} C_VEL
LIN {X 0,Y 530.971,Z 279.339,A -85,B 0,C 180,E1 -4469.355,E2 -4469.355} C_VEL
LIN {X 0,Y 531.012,Z 279.34,A -85,B 0,C 180,E1 -4472.467,E2 -4472.467} C_VEL
LIN {X 0,Y 530.991,Z 279.34,A -85,B 0,C 180,E1 -4474.942,E2 -4474.942} C_VEL
LIN {X 0,Y 530.968,Z 279.343,A -85,B 0,C 180,E1 -4478.247,E2 -4478.247} C_VEL
LIN {X 0,Y 530.993,Z 279.344,A -85,B 0,C 180,E1 -4480.677,E2 -4480.677} C_VEL
LIN {X 0,Y 530.984,Z 279.341,A -85,B 0,C 180,E1 -4483.071,E2 -4483.071} C_VEL
LIN {X 0,Y 531.017,Z 279.335,A -85,B 0,C 180,E1 -4485.436,E2 -4485.436} C_VEL
LIN {X 0,Y 531.034,Z 279.335,A -85,B 0,C 180,E1 -4488.55,E2 -4488.55} C_VEL
LIN {X 0,Y 531.052,Z 279.328,A -85,B 0,C 180,E1 -4491.63,E2 -4491.63} C_VEL
LIN {X 0,Y 531.117,Z 279.328,A -85,B 0,C 180,E1 -4494.685,E2 -4494.685} C_VEL
LIN {X 0,Y 531.138,Z 279.319,A -85,B 0,C 180,E1 -4497.725,E2 -4497.725} C_VEL
LIN {X 0,Y 531.151,Z 279.323,A -85,B 0,C 180,E1 -4500.758,E2 -4500.758} C_VEL
LIN {X 0,Y 531.102,Z 279.331,A -85,B 0,C 180,E1 -4503.034,E2 -4503.034} C_VEL
LIN {X 0,Y 531.08,Z 279.325,A -85,B 0,C 180,E1 -4506.077,E2 -4506.077} C_VEL
LIN {X 0,Y 531.028,Z 279.339,A -85,B 0,C 180,E1 -4509.138,E2 -4509.138} C_VEL
LIN {X 0,Y 531.038,Z 279.331,A -85,B 0,C 180,E1 -4512.225,E2 -4512.225} C_VEL
LIN {X 0,Y 530.994,Z 279.342,A -85,B 0,C 180,E1 -4515.35,E2 -4515.35} C_VEL
LIN {X 0,Y 530.983,Z 279.339,A -85,B 0,C 180,E1 -4518.522,E2 -4518.522} C_VEL
LIN {X 0,Y 530.997,Z 279.343,A -85,B 0,C 180,E1 -4520.938,E2 -4520.938} C_VEL
LIN {X 0,Y 530.96,Z 279.341,A -85,B 0,C 180,E1 -4524.226,E2 -4524.226} C_VEL
LIN {X 0,Y 530.998,Z 279.339,A -85,B 0,C 180,E1 -4526.744,E2 -4526.744} C_VEL
LIN {X 0,Y 530.978,Z 279.347,A -85,B 0,C 180,E1 -4529.323,E2 -4529.323} C_VEL
LIN {X 0,Y 530.963,Z 279.339,A -85,B 0,C 180,E1 -4532.101,E2 -4532.101} C_VEL
LIN {X 0,Y 530.971,Z 279.342,A -85,B 0,C 180,E1 -4534.852,E2 -4534.852} C_VEL
LIN {X 0,Y 530.964,Z 279.345,A -85,B 0,C 180,E1 -4537.508,E2 -4537.508} C_VEL
LIN {X 0,Y 530.963,Z 279.34,A -85,B 0,C 180,E1 -4540.435,E2 -4540.435} C_VEL
LIN {X 0,Y 530.934,Z 279.351,A -85,B 0,C 180,E1 -4543.564,E2 -4543.564} C_VEL
LIN {X 0,Y 530.267,Z 279.43,A -85,B 0,C 180,E1 -4544.197,E2 -4544.197} C_VEL
LIN {X 0,Y 527.423,Z 279.789,A -85,B 0,C 180,E1 -4545.226,E2 -4545.226} C_VEL
LIN {X 0,Y 525.015,Z 280.086,A -85,B 0,C 180,E1 -4546.055,E2 -4546.055} C_VEL
LIN {X 0,Y 523.974,Z 280.214,A -85,B 0,C 180,E1 -4546.694,E2 -4546.694} C_VEL
LIN {X 0,Y 523.885,Z 280.225,A -85,B 0,C 180,E1 -4546.911,E2 -4546.911} C_VEL
LIN {X 0,Y 523.912,Z 280.223,A -85,B 0,C 180,E1 -4549.918,E2 -4549.918} C_VEL
LIN {X 0,Y 523.883,Z 280.225,A -85,B 0,C 180,E1 -4552.866,E2 -4552.866} C_VEL
LIN {X 0,Y 523.919,Z 280.225,A -85,B 0,C 180,E1 -4555.709,E2 -4555.709} C_VEL
LIN {X 0,Y 523.912,Z 280.221,A -85,B 0,C 180,E1 -4558.456,E2 -4558.456} C_VEL
LIN {X 0,Y 523.91,Z 280.226,A -85,B 0,C 180,E1 -4561.124,E2 -4561.124} C_VEL
LIN {X 0,Y 523.978,Z 280.26,A -85,B 0,C 180,E1 -4562.311,E2 -4562.311} C_VEL
LIN {X 0,Y 524.224,Z 285.628,A -85,B 0,C 180,E1 -4563.313,E2 -4563.313} C_VEL
LIN {X 0,Y 524.136,Z 299.493,A -85,B 0,C 180,E1 -4565.888,E2 -4565.888} C_VEL
LIN {X 0,Y 526.023,Z 310.366,A -85,B 0,C 180,E1 -4566.107,E2 -4566.107} C_VEL
LIN {X 0,Y 525.51,Z 406.607,A -85,B 0,C 180,E1 -4567.445,E2 -4567.445} C_VEL
LIN {X 0,Y 525.41,Z 419.872,A -85,B 0,C 180,E1 -4567.791,E2 -4567.791} C_VEL
LIN {X 0,Y 525.135,Z 431.89,A -85,B 0,C 180,E1 -4568.251,E2 -4568.251} C_VEL
LIN {X 0,Y 524.879,Z 444.458,A -85,B 0,C 180,E1 -4568.91,E2 -4568.91} C_VEL
LIN {X 0,Y 524.61,Z 455.778,A -85,B 0,C 180,E1 -4569.681,E2 -4569.681} C_VEL
LIN {X 0,Y 524.31,Z 465.73,A -85,B 0,C 180,E1 -4570.523,E2 -4570.523} C_VEL
LIN {X 0,Y 524.077,Z 474.478,A -85,B 0,C 180,E1 -4571.429,E2 -4571.429} C_VEL
LIN {X 0,Y 523.85,Z 483.257,A -85,B 0,C 180,E1 -4572.548,E2 -4572.548} C_VEL
LIN {X 0,Y 523.65,Z 491.31,A -85,B 0,C 180,E1 -4573.83,E2 -4573.83} C_VEL
LIN {X 0,Y 523.524,Z 497.728,A -85,B 0,C 180,E1 -4575.143,E2 -4575.143} C_VEL
LIN {X 0,Y 523.421,Z 502.469,A -85,B 0,C 180,E1 -4576.41,E2 -4576.41} C_VEL
LIN {X 0,Y 523.36,Z 505.759,A -85,B 0,C 180,E1 -4577.593,E2 -4577.593} C_VEL
LIN {X 0,Y 523.366,Z 507.784,A -85,B 0,C 180,E1 -4578.605,E2 -4578.605} C_VEL
LIN {X 0,Y 523.31,Z 509.346,A -85,B 0,C 180,E1 -4579.946,E2 -4579.946} C_VEL
LIN {X 0,Y 523.34,Z 509.669,A -85,B 0,C 180,E1 -4581.506,E2 -4581.506} C_VEL
LIN {X 0,Y 523.356,Z 509.248,A -85,B 0,C 180,E1 -4582.283,E2 -4582.283} C_VEL
LIN {X 0,Y 523.387,Z 507.662,A -85,B 0,C 180,E1 -4583.552,E2 -4583.552} C_VEL
LIN {X 0,Y 523.357,Z 504.495,A -85,B 0,C 180,E1 -4584.993,E2 -4584.993} C_VEL
LIN {X 0,Y 523.458,Z 500.844,A -85,B 0,C 180,E1 -4586.151,E2 -4586.151} C_VEL
LIN {X 0,Y 523.561,Z 496.1,A -85,B 0,C 180,E1 -4587.308,E2 -4587.308} C_VEL
LIN {X 0,Y 523.71,Z 489.028,A -85,B 0,C 180,E1 -4588.655,E2 -4588.655} C_VEL
LIN {X 0,Y 523.886,Z 481.317,A -85,B 0,C 180,E1 -4589.808,E2 -4589.808} C_VEL
LIN {X 0,Y 524.146,Z 471.721,A -85,B 0,C 180,E1 -4590.961,E2 -4590.961} C_VEL
LIN {X 0,Y 524.366,Z 461.811,A -85,B 0,C 180,E1 -4591.921,E2 -4591.921} C_VEL
LIN {X 0,Y 524.637,Z 450.608,A -85,B 0,C 180,E1 -4592.784,E2 -4592.784} C_VEL
LIN {X 0,Y 524.939,Z 439.634,A -85,B 0,C 180,E1 -4593.454,E2 -4593.454} C_VEL
LIN {X 0,Y 525.132,Z 427.47,A -85,B 0,C 180,E1 -4594.03,E2 -4594.03} C_VEL
LIN {X 0,Y 525.333,Z 414.528,A -85,B 0,C 180,E1 -4594.46,E2 -4594.46} C_VEL
LIN {X 0,Y 525.536,Z 402.054,A -85,B 0,C 180,E1 -4594.723,E2 -4594.723} C_VEL
LIN {X 0,Y 525.922,Z 308.735,A -85,B 0,C 180,E1 -4596.008,E2 -4596.008} C_VEL
LIN {X 0,Y 524.201,Z 299.515,A -85,B 0,C 180,E1 -4596.206,E2 -4596.206} C_VEL
LIN {X 0,Y 524.315,Z 285.499,A -85,B 0,C 180,E1 -4598.868,E2 -4598.868} C_VEL
LIN {X 0,Y 523.902,Z 280.228,A -85,B 0,C 180,E1 -4599.897,E2 -4599.897} C_VEL
LIN {X 0,Y 523.953,Z 280.222,A -85,B 0,C 180,E1 -4602.393,E2 -4602.393} C_VEL
LIN {X 0,Y 523.931,Z 280.216,A -85,B 0,C 180,E1 -4605.562,E2 -4605.562} C_VEL
LIN {X 0,Y 523.917,Z 280.218,A -85,B 0,C 180,E1 -4607.971,E2 -4607.971} C_VEL
LIN {X 0,Y 523.958,Z 280.217,A -85,B 0,C 180,E1 -4610.411,E2 -4610.411} C_VEL
LIN {X 0,Y 523.913,Z 280.227,A -85,B 0,C 180,E1 -4612.894,E2 -4612.894} C_VEL
LIN {X 0,Y 523.9,Z 280.222,A -85,B 0,C 180,E1 -4615.422,E2 -4615.422} C_VEL
LIN {X 0,Y 523.906,Z 280.219,A -85,B 0,C 180,E1 -4618.003,E2 -4618.003} C_VEL
LIN {X 0,Y 523.905,Z 280.227,A -85,B 0,C 180,E1 -4620.846,E2 -4620.846} C_VEL
LIN {X 0,Y 523.932,Z 280.217,A -85,B 0,C 180,E1 -4623.729,E2 -4623.729} C_VEL
LIN {X 0,Y 523.903,Z 280.22,A -85,B 0,C 180,E1 -4626.4,E2 -4626.4} C_VEL
LIN {X 0,Y 523.915,Z 280.226,A -85,B 0,C 180,E1 -4629.086,E2 -4629.086} C_VEL
LIN {X 0,Y 523.898,Z 280.22,A -85,B 0,C 180,E1 -4632.125,E2 -4632.125} C_VEL
LIN {X 0,Y 523.939,Z 280.225,A -85,B 0,C 180,E1 -4635.311,E2 -4635.311} C_VEL
LIN {X 0,Y 523.919,Z 280.218,A -85,B 0,C 180,E1 -4638.695,E2 -4638.695} C_VEL
LIN {X 0,Y 523.906,Z 280.222,A -85,B 0,C 180,E1 -4641.897,E2 -4641.897} C_VEL
LIN {X 0,Y 523.923,Z 280.218,A -85,B 0,C 180,E1 -4644.912,E2 -4644.912} C_VEL
LIN {X 0,Y 523.94,Z 280.223,A -85,B 0,C 180,E1 -4647.68,E2 -4647.68} C_VEL
LIN {X 0,Y 523.957,Z 280.213,A -85,B 0,C 180,E1 -4650.677,E2 -4650.677} C_VEL
LIN {X 0,Y 523.895,Z 280.231,A -85,B 0,C 180,E1 -4653.724,E2 -4653.724} C_VEL
LIN {X 0,Y 523.913,Z 280.221,A -85,B 0,C 180,E1 -4656.269,E2 -4656.269} C_VEL
LIN {X 0,Y 523.95,Z 280.214,A -85,B 0,C 180,E1 -4658.766,E2 -4658.766} C_VEL
LIN {X 0,Y 523.938,Z 280.216,A -85,B 0,C 180,E1 -4661.22,E2 -4661.22} C_VEL
LIN {X 0,Y 523.907,Z 280.224,A -85,B 0,C 180,E1 -4663.638,E2 -4663.638} C_VEL
LIN {X 0,Y 523.929,Z 280.226,A -85,B 0,C 180,E1 -4666.027,E2 -4666.027} C_VEL
LIN {X 0,Y 523.964,Z 280.216,A -85,B 0,C 180,E1 -4668.393,E2 -4668.393} C_VEL
LIN {X 0,Y 523.957,Z 280.214,A -85,B 0,C 180,E1 -4671.515,E2 -4671.515} C_VEL
LIN {X 0,Y 524.035,Z 280.206,A -85,B 0,C 180,E1 -4674.613,E2 -4674.613} C_VEL
LIN {X 0,Y 524.107,Z 280.196,A -85,B 0,C 180,E1 -4677.694,E2 -4677.694} C_VEL
LIN {X 0,Y 524.076,Z 280.201,A -85,B 0,C 180,E1 -4680.768,E2 -4680.768} C_VEL
LIN {X 0,Y 524,Z 280.208,A -85,B 0,C 180,E1 -4683.075,E2 -4683.075} C_VEL
LIN {X 0,Y 524.007,Z 280.212,A -85,B 0,C 180,E1 -4686.159,E2 -4686.159} C_VEL
LIN {X 0,Y 523.946,Z 280.215,A -85,B 0,C 180,E1 -4689.263,E2 -4689.263} C_VEL
LIN {X 0,Y 523.951,Z 280.221,A -85,B 0,C 180,E1 -4692.393,E2 -4692.393} C_VEL
LIN {X 0,Y 523.928,Z 280.216,A -85,B 0,C 180,E1 -4695.562,E2 -4695.562} C_VEL
LIN {X 0,Y 523.915,Z 280.219,A -85,B 0,C 180,E1 -4697.971,E2 -4697.971} C_VEL
LIN {X 0,Y 523.955,Z 280.218,A -85,B 0,C 180,E1 -4700.411,E2 -4700.411} C_VEL
LIN {X 0,Y 523.911,Z 280.227,A -85,B 0,C 180,E1 -4702.894,E2 -4702.894} C_VEL
LIN {X 0,Y 523.897,Z 280.222,A -85,B 0,C 180,E1 -4705.422,E2 -4705.422} C_VEL
LIN {X 0,Y 523.903,Z 280.219,A -85,B 0,C 180,E1 -4708.003,E2 -4708.003} C_VEL
LIN {X 0,Y 523.903,Z 280.227,A -85,B 0,C 180,E1 -4710.846,E2 -4710.846} C_VEL
LIN {X 0,Y 523.929,Z 280.217,A -85,B 0,C 180,E1 -4713.729,E2 -4713.729} C_VEL
LIN {X 0,Y 523.901,Z 280.221,A -85,B 0,C 180,E1 -4716.4,E2 -4716.4} C_VEL
LIN {X 0,Y 523.913,Z 280.227,A -85,B 0,C 180,E1 -4719.086,E2 -4719.086} C_VEL
LIN {X 0,Y 523.895,Z 280.22,A -85,B 0,C 180,E1 -4722.125,E2 -4722.125} C_VEL
LIN {X 0,Y 523.937,Z 280.225,A -85,B 0,C 180,E1 -4725.311,E2 -4725.311} C_VEL
LIN {X 0,Y 523.917,Z 280.219,A -85,B 0,C 180,E1 -4728.695,E2 -4728.695} C_VEL
LIN {X 0,Y 523.904,Z 280.222,A -85,B 0,C 180,E1 -4731.897,E2 -4731.897} C_VEL
LIN {X 0,Y 523.921,Z 280.219,A -85,B 0,C 180,E1 -4734.912,E2 -4734.912} C_VEL
LIN {X 0,Y 523.938,Z 280.224,A -85,B 0,C 180,E1 -4737.68,E2 -4737.68} C_VEL
LIN {X 0,Y 523.955,Z 280.214,A -85,B 0,C 180,E1 -4740.677,E2 -4740.677} C_VEL
LIN {X 0,Y 523.893,Z 280.23,A -85,B 0,C 180,E1 -4743.724,E2 -4743.724} C_VEL
LIN {X 0,Y 523.938,Z 280.231,A -85,B 0,C 180,E1 -4745.005,E2 -4745.005} C_VEL
LIN {X 0,Y 525.471,Z 288.481,A -85,B 0,C 180,E1 -4746.344,E2 -4746.344} C_VEL
LIN {X 0,Y 525.115,Z 306.108,A -85,B 0,C 180,E1 -4749.021,E2 -4749.021} C_VEL
LIN {X 0,Y 524.642,Z 326.389,A -85,B 0,C 180,E1 -4752.055,E2 -4752.055} C_VEL
LIN {X 0,Y 524.31,Z 345.34,A -85,B 0,C 180,E1 -4754.842,E2 -4754.842} C_VEL
LIN {X 0,Y 525.895,Z 356.428,A -85,B 0,C 180,E1 -4755.041,E2 -4755.041} C_VEL
LIN {X 0,Y 525.474,Z 453.721,A -85,B 0,C 180,E1 -4756.39,E2 -4756.39} C_VEL
LIN {X 0,Y 525.248,Z 467.048,A -85,B 0,C 180,E1 -4756.729,E2 -4756.729} C_VEL
LIN {X 0,Y 525.002,Z 479.251,A -85,B 0,C 180,E1 -4757.19,E2 -4757.19} C_VEL
LIN {X 0,Y 524.778,Z 491.331,A -85,B 0,C 180,E1 -4757.808,E2 -4757.808} C_VEL
LIN {X 0,Y 524.503,Z 503.203,A -85,B 0,C 180,E1 -4758.6,E2 -4758.6} C_VEL
LIN {X 0,Y 524.207,Z 513.678,A -85,B 0,C 180,E1 -4759.474,E2 -4759.474} C_VEL
LIN {X 0,Y 523.985,Z 522.247,A -85,B 0,C 180,E1 -4760.348,E2 -4760.348} C_VEL
LIN {X 0,Y 523.779,Z 530.155,A -85,B 0,C 180,E1 -4761.317,E2 -4761.317} C_VEL
LIN {X 0,Y 523.603,Z 537.88,A -85,B 0,C 180,E1 -4762.48,E2 -4762.48} C_VEL
LIN {X 0,Y 523.48,Z 545.004,A -85,B 0,C 180,E1 -4763.834,E2 -4763.834} C_VEL
LIN {X 0,Y 523.384,Z 549.742,A -85,B 0,C 180,E1 -4764.992,E2 -4764.992} C_VEL
LIN {X 0,Y 523.443,Z 553.369,A -85,B 0,C 180,E1 -4766.15,E2 -4766.15} C_VEL
LIN {X 0,Y 523.367,Z 555.234,A -85,B 0,C 180,E1 -4766.92,E2 -4766.92} C_VEL
LIN {X 0,Y 523.334,Z 556.634,A -85,B 0,C 180,E1 -4767.691,E2 -4767.691} C_VEL
LIN {X 0,Y 523.252,Z 558.241,A -85,B 0,C 180,E1 -4769.23,E2 -4769.23} C_VEL
LIN {X 0,Y 523.254,Z 558.458,A -85,B 0,C 180,E1 -4770,E2 -4770} C_VEL
LIN {X 0,Y 523.274,Z 557.632,A -85,B 0,C 180,E1 -4771.539,E2 -4771.539} C_VEL
LIN {X 0,Y 523.334,Z 556.635,A -85,B 0,C 180,E1 -4772.308,E2 -4772.308} C_VEL
LIN {X 0,Y 523.367,Z 555.235,A -85,B 0,C 180,E1 -4773.079,E2 -4773.079} C_VEL
LIN {X 0,Y 523.424,Z 552.29,A -85,B 0,C 180,E1 -4774.235,E2 -4774.235} C_VEL
LIN {X 0,Y 523.461,Z 548.3,A -85,B 0,C 180,E1 -4775.392,E2 -4775.392} C_VEL
LIN {X 0,Y 523.513,Z 543.072,A -85,B 0,C 180,E1 -4776.571,E2 -4776.571} C_VEL
LIN {X 0,Y 523.638,Z 536.706,A -85,B 0,C 180,E1 -4777.713,E2 -4777.713} C_VEL
LIN {X 0,Y 523.819,Z 528.65,A -85,B 0,C 180,E1 -4778.875,E2 -4778.875} C_VEL
LIN {X 0,Y 524.015,Z 520.441,A -85,B 0,C 180,E1 -4779.846,E2 -4779.846} C_VEL
LIN {X 0,Y 524.271,Z 510.436,A -85,B 0,C 180,E1 -4780.817,E2 -4780.817} C_VEL
LIN {X 0,Y 524.625,Z 499.132,A -85,B 0,C 180,E1 -4781.691,E2 -4781.691} C_VEL
LIN {X 0,Y 524.842,Z 488.085,A -85,B 0,C 180,E1 -4782.371,E2 -4782.371} C_VEL
LIN {X 0,Y 525.074,Z 475.831,A -85,B 0,C 180,E1 -4782.955,E2 -4782.955} C_VEL
LIN {X 0,Y 525.348,Z 462.982,A -85,B 0,C 180,E1 -4783.391,E2 -4783.391} C_VEL
LIN {X 0,Y 525.516,Z 450.865,A -85,B 0,C 180,E1 -4783.658,E2 -4783.658} C_VEL
LIN {X 0,Y 525.803,Z 355.147,A -85,B 0,C 180,E1 -4784.979,E2 -4784.979} C_VEL
LIN {X 0,Y 524.3,Z 345.077,A -85,B 0,C 180,E1 -4785.175,E2 -4785.175} C_VEL
LIN {X 0,Y 524.74,Z 322.358,A -85,B 0,C 180,E1 -4788.527,E2 -4788.527} C_VEL
LIN {X 0,Y 525.085,Z 304.558,A -85,B 0,C 180,E1 -4791.185,E2 -4791.185} C_VEL
